METHOD WriteError
VAR_INPUT
	Event			: E_Event;
	Description 	: T_MaxString;
END_VAR
WriteEvent(ePriority_fault, Event, Description, TRUE);
//eState := E_ComponentState.eComponentState_error;
END_METHOD

METHOD WriteEvent
VAR_INPUT
	Priority		: E_Priority;
	Event			: E_Event;
	Description 	: T_MaxString;
	Signalize			: BOOL;
END_VAR
VAR
	tmpItem: ST_Event;
END_VAR
// chk
IF NOT __ISVALIDREF(fbEventLog) THEN
	RETURN;
END_IF

tmpItem.eComponent := eTyp;
tmpItem.eEventID := Event;
tmpItem.eMachineArea := eMachineArea;
tmpItem.ePriority := Priority;
tmpItem.nComponentID := iId;
tmpItem.sDescription := Description;
tmpItem.bSignalize := Signalize;

IF 	ptLastEvent <> 0 AND_THEN
	ptLastEvent^.bIsRaised AND_THEN
   	tmpItem.eEventID = ptLastEvent^.eEventID AND_THEN
	tmpItem.sDescription = ptLastEvent^.sDescription AND_THEN 
	tmpItem.ePriority = ptLastEvent^.ePriority THEN 
	RETURN;
END_IF

ptLastEvent := fbEventLog.SetEvent(tmpItem);
stLastEvent := tmpItem;
END_METHOD

METHOD WriteInfo
VAR_INPUT
	Event			: E_Event;
	Description 	: T_MaxString;
END_VAR
WriteEvent(ePriority_info, Event, Description, FALSE);
END_METHOD

METHOD WriteWarning
VAR_INPUT
	Event			: E_Event;
	Description 	: T_MaxString;
	Signal			: BOOL;
END_VAR
VAR
	tmpItem			: ST_Event;
END_VAR
WriteEvent(ePriority_warning, Event, Description, Signal);
END_METHOD

END_FUNCTION_BLOCK

// ---- BaseComponents/EventLog/FB_EventLog.TcPOU
/// HMI access provider (host for sub hmi provider)
FUNCTION_BLOCK  FB_EventLog
VAR	
	/// interfaces
	ILog						: ITFLoggingProvider;
	stLogConfig					: ST_LoggingConfig;
	
	/// Logging Provider
	fbDebugLog					: FB_DebugLoggingProvider;
	fbFileLog					: FB_FileLoggingProvider;
	fbEventLog					: FB_EventLoggingProvider;	
	fbEventlogger 				: FB_TcEventLogger;


	/// default notification array mirror (for compare)
	aEvents						: ARRAY[0..iMaxIdxEvents] OF ST_Event;
	aEventsMirror				: ARRAY[0..iMaxIdxEvents] OF ST_Event;
	diEventsChanged				: DINT;	
	diEventsChangedOld			: DINT;	
	nLastIndex					: INT;
	
	ptLastEvent					: POINTER TO ST_Event;
	
	//aEventsMirror				: ARRAY[0..iMaxIdxMachineAreas, 0..iMaxIdxComponent, 0..iMaxIdxEvents] OF ST_Event;
	/// private var's
	eErrorLevel					: E_Priority;
	eErrorLevelMirror			: E_Priority;	
	eLogLevel					: E_LogLevel;	
	
	bMute						: BOOL;
	
	fbAlarm						: FB_TcAlarm;
	fbMessage					: FB_TcMessage;
END_VAR

///
/// Event Log
/// Hannes Fuger /www.asma.at/01.2016
///

PROPERTY Config : ST_LoggingConfig
GET
Config := stLogConfig;
END_GET
SET
stLogConfig := Config;
END_SET
END_PROPERTY

/// System error level
PROPERTY ErrorLevel : E_Priority
GET // INTERNAL
ErrorLevel := eErrorLevel;
END_GET
END_PROPERTY

PROPERTY EventsChanged : BOOL
GET
EventsChanged := diEventsChanged <> diEventsChangedOld;
END_GET
END_PROPERTY

/// Filtert aktuelle Meldungen
METHOD PUBLIC FilterEvents : BOOL
VAR_INPUT
	/// Notification filter
	stFilter	: ST_EventFilter;
END_VAR
VAR_IN_OUT
	/// notification array (result)
	aResult		: ARRAY[0..iMaxIdxEvents] OF ST_Event;
END_VAR
VAR
	idx, iRes, iLast 		: INT;
	bFilterOk				: BOOL;
END_VAR
iRes := 0;
MEMSET(ADR(aResult), 0, SIZEOF(aResult));
iLast := nLastIndex+1;

FOR idx := 0 TO iMaxIdxEvents DO
	bFilterOk := TRUE;
	// IsRaised - Filter
	IF (stFilter.eIsRaisedFilter = eBoolFilter_false AND aEvents[iLast].bIsRaised) OR_ELSE 
	   (stFilter.eIsRaisedFilter = eBoolFilter_true AND NOT aEvents[iLast].bIsRaised) THEN
		bFilterOk := FALSE;
	END_IF
	
	// Area - Filter
	IF (stFilter.eAreaFilter <> E_MachineArea.eMachineArea_none) AND_THEN
	   (stFilter.eAreaFilter <> aEvents[iLast].eMachineArea) THEN
		bFilterOk := FALSE;
	END_IF
	
	// Error - Filter
	IF bFilterOk AND ((stFilter.eErrorFilter AND (aEvents[iLast].ePriority = ePriority_fault OR aEvents[iLast].ePriority = ePriority_faultEmergency OR aEvents[iLast].ePriority = ePriority_faultFastStop))
	// Warning - Filter
	OR (stFilter.eWarningFilter AND aEvents[iLast].ePriority = E_Priority.ePriority_warning)	
	// Info - Filter
	OR (stFilter.eInfoFilter AND aEvents[iLast].ePriority = E_Priority.ePriority_info)) THEN
		
		// add notification to result
		MEMCPY(ADR(aResult[iRes]), ADR(aEvents[iLast]), SIZEOF(aEvents[iLast]));
		iRes := iRes + 1;
	END_IF
	iLast := (iLast+1) MOD (iMaxIdxEvents+1);	
END_FOR

IF iRes > 0 THEN
	FilterEvents := TRUE;
END_IF
END_METHOD

PROPERTY LastIndex : INT
GET
LastIndex := nLastIndex;
END_GET
END_PROPERTY

PROPERTY Logger : REFERENCE TO ITFLoggingProvider
GET
Logger REF= ILog;
END_GET
END_PROPERTY

PROPERTY Mute : BOOL
GET
Mute := bMute;
END_GET
SET
bMute := Mute;
END_SET
END_PROPERTY

PROPERTY NextIndex : INT
GET
NextIndex := (nLastIndex+1) MOD (iMaxIdxEvents+1);
END_GET
END_PROPERTY

/// sets the corresponding notification item flag raised
{attribute 'object_name' := 'QuittAll'}
METHOD QuittAll
VAR_INPUT
	eMachineArea	: E_MachineArea;
END_VAR
VAR
	ni				: INT;
END_VAR
FOR ni := 0 TO iMaxIdxEvents DO	
	IF NOT aEvents[ni].bIsRaised THEN
		CONTINUE;
	END_IF
	
	IF aEvents[ni].eMachineArea = eMachineArea OR eMachineArea = E_MachineArea.eMachineArea_none THEN
		QuittEvent(	aEvents[ni]);
	END_IF
END_FOR
END_METHOD

/// sets the corresponding notification item flag raised
{attribute 'object_name' := 'QuittEvent'}
METHOD QuittEvent
VAR_INPUT
	stItem			: ST_Event;
END_VAR
VAR
	ni				: INT;
	cmpItem			: ST_Event;
END_VAR
// suchen ob ähnlicher Eintrag vorhanden 
// auch diesen quittieren

FOR ni := 0 TO iMaxIdxEvents DO	
	IF aEvents[ni].bIsRaised THEN
		cmpItem := 	aEvents[ni];
		// gleichsetzen damit beim Cmp kein Unterschied bei diesen Werten
		cmpItem.dtQuitTime := stItem.dtQuitTime;			
		cmpItem.dtRaiseTime := stItem.dtRaiseTime;	
		cmpItem.nIdx := stItem.nIdx;	
		
		IF MEMCMP(ADR(cmpItem), ADR(stItem), SIZEOF(ST_EVENT)) = 0 THEN
			aEvents[ni].bIsRaised := FALSE;
			aEvents[ni].dtQuitTime := Statics.dtNow;
			aEvents[ni].sQuitTime := SEL(aEvents[ni].dtQuitTime = DT#1970-01-01-00:00:00, REPLACE(DT_TO_STRING(aEvents[ni].dtQuitTime), '', 3, 1), '');		
		END_IF
		
	END_IF
END_FOR
END_METHOD

/// resets all notification flags and reset-needed state 
{attribute '' := ''}
{attribute 'object_name' := 'Reset'}
METHOD Reset
VAR
	ii: INT;
END_VAR
// reset all items in default notification array
MEMSET(ADR(aEvents), 0, SIZEOF(aEvents));
MEMSET(ADR(aEventsMirror), 0, SIZEOF(aEventsMirror));

// set default message priority
FOR ii := 0 TO iMaxIdxEvents DO
	aEvents[ii].ePriority := E_Priority.ePriority_fault;
END_FOR

nLastIndex := -1;

eErrorLevel			:= ePriority_none;
eErrorLevelMirror	:= ePriority_none;
eLogLevel			:= eLogLevelNone;

// set up logging provider
IF stLogConfig.eLoggingProvider = eLoggingProviderFile THEN
	fbFileLog(stLogConfig := stLogConfig);
	ILog := fbFileLog;
ELSIF stLogConfig.eLoggingProvider = eLoggingProviderEventLog THEN
	fbEventLog(stLogConfig := stLogConfig);
	ILog := fbEventLog;
ELSE // default
	ILog := fbDebugLog;
END_IF
END_METHOD

METHOD Run : E_ComponentState
VAR	/// private variabe
	ii			: INT;	
END_VAR
// run Logger
IF ILog <> 0 THEN
	ILog.Run();
END_IF

diEventsChangedOld := diEventsChanged;
// trigger notification changes
IF (MEMCMP(ADR(aEventsMirror), ADR(aEvents), SIZEOF(aEvents)) <> 0) THEN
	diEventsChanged := diEventsChanged  + 1; // in case of index-overrun, it (re)starts itself (-DINT max)
	aEventsMirror := aEvents;
END_IF

// get max error level
eErrorLevel := E_Priority.ePriority_none;
FOR ii := 0 TO iMaxIdxEvents DO	
	IF aEvents[ii].bIsRaised THEN
		eErrorLevel := MAX(eErrorLevel, aEvents[ii].ePriority);
		IF eErrorLevel <> eErrorLevelMirror THEN
			eErrorLevelMirror := eErrorLevel;
			CASE eErrorLevel OF
				E_Priority.ePriority_none,
				E_Priority.ePriority_info:
					eLogLevel := E_Loglevel.eLogLevelInformation;
				E_Priority.ePriority_warning:
					eLogLevel := E_Loglevel.eLogLevelWarning;
				E_Priority.ePriority_fault,
				E_Priority.ePriority_faultFastStop,
				E_Priority.ePriority_faultEmergency:
					eLogLevel := E_Loglevel.eLogLevelError;
			END_CASE
			ILog.AddLog(Concat6('ErrorLevel changed, ID: ', INT_TO_STRING(aEvents[ii].nComponentID),'-',INT_TO_STRING(aEvents[ii].eEventID),', MSG: ', aEvents[ii].sDescription), 'Supervision', eLogLevel);
		END_IF
	END_IF
END_FOR
END_METHOD

/// sets the corresponding notification item flag raised
{attribute 'object_name' := 'SetEvent'}
METHOD SetEvent : POINTER TO ST_Event
VAR_INPUT
	/// item to set
	stItem: ST_Event;
END_VAR
VAR
	tmpIndex		: INT;
	cmpItem			: ST_Event;
END_VAR
// suchen ob Eintrag schon vorhanden 
// nach gewisser zeit wieder eintragen
// sonst nichts unterenheme

// set item in default notification array 
tmpIndex := nextIndex;

// letzter Event der selbe?
IF tmpIndex > 0 THEN
	cmpItem := aEvents[LastIndex];
	// gleichsetzen damit beim Cmp kein Unterschied bei diesen Werten
	cmpItem.dtQuitTime := stItem.dtQuitTime;
	cmpItem.dtRaiseTime := stItem.dtRaiseTime;
	cmpItem.nIdx := stItem.nIdx;
	
	IF MEMCMP(ADR(stItem), ADR(cmpItem), SIZEOF(ST_Event)) = 0 THEN 
		RETURN;
	END_IF
END_IF


aEvents[tmpIndex] := stItem;
aEvents[tmpIndex].nIdx := tmpIndex;
aEvents[tmpIndex].bIsRaised := TRUE;
aEvents[tmpIndex].dtRaiseTime := Statics.dtNow;
aEvents[tmpIndex].dtQuitTime := StaticsConstant.dtMinValue;

aEvents[tmpIndex].sRaiseTime := SEL(aEvents[tmpIndex].dtRaiseTime = DT#1970-01-01-00:00:00, REPLACE(DT_TO_STRING(aEvents[tmpIndex].dtRaiseTime), '', 3, 1), '');
aEvents[tmpIndex].sQuitTime := SEL(aEvents[tmpIndex].dtQuitTime = DT#1970-01-01-00:00:00, REPLACE(DT_TO_STRING(aEvents[tmpIndex].dtQuitTime), '', 3, 1), '');

nLastIndex := tmpIndex;
SetEvent := ADR(aEvents[nLastIndex]);
END_METHOD

METHOD WriteError
VAR_INPUT
	Event			: E_Event;
	Description 	: T_MaxString;
END_VAR
WriteEvent(ePriority_fault, Event, Description, TRUE);
//eState := E_ComponentState.eComponentState_error;
END_METHOD

METHOD WriteEvent
VAR_INPUT
	Priority		: E_Priority;
	Event			: E_Event;
	Description 	: T_MaxString;
	Signalize		: BOOL;
END_VAR
VAR
	tmpItem			: ST_Event;
END_VAR
// chk

tmpItem.eComponent := E_ComponentType.eComponentType_none;
tmpItem.eEventID := Event;
tmpItem.eMachineArea := E_MachineArea.eMachineArea_common;
tmpItem.ePriority := Priority;
tmpItem.nComponentID := 0;
tmpItem.sDescription := Description;
tmpItem.bSignalize := Signalize;

IF 	ptLastEvent <> 0 AND_THEN
	ptLastEvent^.bIsRaised AND_THEN
   	tmpItem.eEventID = ptLastEvent^.eEventID AND_THEN
	tmpItem.sDescription = ptLastEvent^.sDescription AND_THEN 
	tmpItem.ePriority = ptLastEvent^.ePriority THEN 
	RETURN;
END_IF

ptLastEvent := SetEvent(tmpItem);
END_METHOD

METHOD WriteInfo
VAR_INPUT
	Event			: E_Event;
	Description 	: T_MaxString;
END_VAR
WriteEvent(ePriority_info, Event, Description, FALSE);
END_METHOD

METHOD WriteWarning
VAR_INPUT
	Event			: E_Event;
	Description 	: T_MaxString;
	Signal			: BOOL;
END_VAR
VAR
	tmpItem			: ST_Event;
END_VAR
WriteEvent(ePriority_warning, Event, Description, Signal);
END_METHOD

END_FUNCTION_BLOCK

// ---- Visualisation/P_Visu.TcPOU
PROGRAM P_Visu
VAR
	bFirstRun					: BOOL := TRUE;	
	
END_VAR

IF bFirstRun THEN
	bFirstRun := FALSE;
	FirstRun();
END_IF

JogButton();
SwitchButton();
SyncVariable();

METHOD FirstRun : BOOL
VAR_INPUT
END_VAR
GVL_VISU.stMachineConfig := P_Machine.MachineConfig;	
GVL_VISU.stCurMat := fbmat.Mat;
END_METHOD

METHOD JogButton : BOOL
VAR_INPUT
END_VAR
// JOG X
IF GVL_VISU.stMaintCmds.bJogXBw THEN
	GVL.fbMatAndToolHandling.JogX(TRUE);
ELSIF GVL_VISU.stMaintCmds.bJogXFw THEN
	GVL.fbMatAndToolHandling.JogX(FALSE);
ELSE
	GVL.fbMatAndToolHandling.JogXStop();
END_IF

// JOG Y
IF GVL_VISU.stMaintCmds.bJogYBw THEN
	GVL.fbMatAndToolHandling.JogY(TRUE);
ELSIF GVL_VISU.stMaintCmds.bJogYFw THEN
	GVL.fbMatAndToolHandling.JogY(FALSE);
ELSE
	GVL.fbMatAndToolHandling.JogYStop();
END_IF

// JOG Punch
IF GVL_VISU.stMaintCmds.bJogPunchBw THEN
	GVL.fbPunchEngine.Jog(FALSE, TRUE);
ELSIF GVL_VISU.stMaintCmds.bJogPunchFw THEN
	GVL.fbPunchEngine.Jog(TRUE, FALSE);
ELSE
	GVL.fbPunchEngine.JogStop();
END_IF

// JOG BELT
IF GVL_VISU.stMaintCmds.bJogOutletBelt THEN
	GVL.fbPunchEngine.OutletBeltJog(TRUE);
ELSE
	GVL.fbPunchEngine.OutletBeltJog(FALSE);
END_IF
END_METHOD

METHOD SwitchButton : BOOL
VAR_STAT
	stNullPunchCmds				: ST_PunchCmds;
	stNullMaintCmds				: ST_MaintCmds;
END_VAR
// PUNCH COMMANDS
IF MEMCMP(ADR(GVL_VISU.stPunchCmds), ADR(stNullPunchCmds), SIZEOF(ST_PunchCmds)) <> 0 THEN
	IF GVL_VISU.stPunchCmds.bLoad THEN
		P_Machine.LoadMat(GVL_VISU.stCurMat);		
		P_Machine.LoadJob(GVL_VISU.stPunchJob);	
	END_IF
	
	IF GVL_VISU.stPunchCmds.bStart THEN	
		P_Machine.LoadMat(GVL_VISU.stCurMat);	
		P_Machine.Start(GVL_VISU.stPunchJob);	
	END_IF
	
	IF GVL_VISU.stPunchCmds.bStop THEN
		P_Machine.Stop();	
	END_IF
	
	IF GVL_VISU.stPunchCmds.bResume THEN
		P_Machine.Resume();	
	END_IF
	
	IF GVL_VISU.stPunchCmds.bHalt THEN
		P_Machine.ClearJob();
		P_Machine.Halt();	
	END_IF	
		
	IF GVL_VISU.stPunchCmds.bLoadLeft THEN
		P_Machine.Maint(TRUE, TRUE, FALSE);	
	END_IF	
	
	IF GVL_VISU.stPunchCmds.bLoadRight THEN
		P_Machine.Maint(TRUE, TRUE, TRUE);	
	END_IF	
	
	IF GVL_VISU.stPunchCmds.bLoadStop THEN
		P_Machine.Halt();	
	END_IF	
	
	IF GVL_VISU.stPunchCmds.bUnlock THEN
		IF fbSafetyLock.Locked THEN
			GVL.fbSafetyLock.Unlock();
		ELSE
			GVL.fbSafetyLock.Lock();
		END_IF
	END_IF		
	
	IF GVL_VISU.stPunchCmds.bMoveTDC THEN
		GVL.fbPunchEngine.MoveTDC();	
	END_IF	
	
	IF GVL_VISU.stPunchCmds.bOutletBelt THEN
		GVL.fbPunchEngine.OutletBeltOnce();	
	END_IF	
		
	IF GVL_VISU.stPunchCmds.bOverride THEN
		P_Machine.Override := GVL_VISU.stPunchParam.fOverride;
	END_IF	
END_IF

// RESET PUNCH COMMANDS
GVL_VISU.stPunchCmds.bLoad := FALSE;
GVL_VISU.stPunchCmds.bStart := FALSE;
GVL_VISU.stPunchCmds.bStop := FALSE;
GVL_VISU.stPunchCmds.bResume := FALSE;
GVL_VISU.stPunchCmds.bHalt := FALSE;
GVL_VISU.stPunchCmds.bLoadLeft := FALSE;
GVL_VISU.stPunchCmds.bLoadRight := FALSE;
GVL_VISU.stPunchCmds.bMoveTDC := FALSE;
GVL_VISU.stPunchCmds.bOutletBelt := FALSE;
GVL_VISU.stPunchCmds.bOverride := FALSE;
GVL_VISU.stPunchCmds.bUnlock := FALSE;
GVL_VISU.stPunchCmds.bLoadStop := FALSE;

// MAINT COMMANDS
IF MEMCMP(ADR(GVL_VISU.stMaintCmds), ADR(stNullMaintCmds), SIZEOF(ST_MaintCmds)) <> 0 THEN	
	IF GVL_VISU.stMaintCmds.bLoadConfig THEN
		P_Machine.LoadConfig(GVL_VISU.stMachineConfig);
	END_IF
	
	IF GVL_VISU.stMaintCmds.bChangeTool THEN
		GVL.fbMatAndToolHandling.ChangeTool(GVL_VISU.stMaintParam.nChangeTool);
	END_IF
	
	IF GVL_VISU.stMaintCmds.bMoveXYMaint THEN
		P_Machine.Maint(TRUE, TRUE, FALSE);	
	END_IF
	
	IF GVL_VISU.stMaintCmds.bMoveXYMaintAlt THEN
		P_Machine.Maint(TRUE, TRUE, TRUE);	
	END_IF
	
	IF GVL_VISU.stMaintCmds.bReset THEN
		P_Machine.Reset();	
	END_IF	
	
	IF GVL_VISU.stMaintCmds.bMovePunchTDC THEN
		GVL.fbPunchEngine.MoveTDC();	
	END_IF	
	
	IF GVL_VISU.stMaintCmds.bSetZero THEN
		GVL.fbPunchEngine.SetZeroOffset();	
	END_IF	
	
END_IF

// RESET MAINT COMMANDS
GVL_VISU.stMaintCmds.bLoadConfig := FALSE;
GVL_VISU.stMaintCmds.bChangeTool := FALSE;
GVL_VISU.stMaintCmds.bMoveXYMaint := FALSE;
GVL_VISU.stMaintCmds.bMoveXYMaintAlt := FALSE;
GVL_VISU.stMaintCmds.bReset := FALSE;
GVL_VISU.stMaintCmds.bMovePunchTDC := FALSE; 
GVL_VISU.stMaintCmds.bSetZero := FALSE;
END_METHOD

METHOD SyncVariable : BOOL
VAR_INPUT
END_VAR
// VISU TO PLC
stPunchInfo.sCleartext 				:= P_Machine.seqOpMode.ClearText;
stPunchInfo.nCurMat 				:= P_Machine.CurMat + 1;
stPunchInfo.nCurPunch 				:= P_Machine.CurPunch + 1;
stPunchInfo.nCurRun 				:= P_Machine.CurRun + 1;
stPunchInfo.nMaxPunches 			:= P_Machine.MaxPunch + 1;
stPunchInfo.nCountRemainHolesOfJob 	:= P_Machine.CountRemainHolesOfJob + 1;
stPunchInfo.nCountAllHolesOfJob 	:= P_Machine.CountAllHolesOfJob + 1;
stPunchInfo.nRemainTimeOfJob 		:= P_Machine.RemainTimeOfJob;
stPunchInfo.stCoordinate 			:= P_Machine.stCoordinate;
stPunchInfo.bPunching 				:= P_Machine.Punching;
stPunchInfo.bResumeAllowed 			:= P_Machine.ResumeAllowed;
stPunchInfo.eJobState 				:= P_Machine.JobState;
stPunchInfo.fOverride 				:= P_Machine.Override;
stPunchInfo.fPunchspeed				:= fbPunchEngine.fbPunchAxis.Velocity;
stPunchInfo.bLocked					:= fbSafetyLock.Locked;

// X - Axis
stMaintInfo.bXHomed					:= fbMatAndToolHandling.fbAxisX.Homed;
stMaintInfo.bXError					:= fbMatAndToolHandling.fbAxisX.Error;
stMaintInfo.bXMoving				:= fbMatAndToolHandling.fbAxisX.Moving;
stMaintInfo.fXPosition				:= fbMatAndToolHandling.fbAxisX.ActPos;
stMaintInfo.fXTemp					:= fbMatAndToolHandling.fbAxisX.AmplifierTemp;
stMaintInfo.fXMotorTemp				:= fbMatAndToolHandling.fbAxisX.MotorTemp;
                            		   
// Y - Axis                 		   
stMaintInfo.bYHomed					:= fbMatAndToolHandling.fbAxisY.Homed;        
stMaintInfo.bYError					:= fbMatAndToolHandling.fbAxisY.Error;        
stMaintInfo.bYMoving				:= fbMatAndToolHandling.fbAxisY.Moving;       
stMaintInfo.fYPosition				:= fbMatAndToolHandling.fbAxisY.ActPos;       
stMaintInfo.fYTemp					:= fbMatAndToolHandling.fbAxisY.AmplifierTemp;
stMaintInfo.fYMotorTemp				:= fbMatAndToolHandling.fbAxisY.MotorTemp;    
                            		   
// Punch - Axis             		   
stMaintInfo.bPunchHomed				:= fbPunchEngine.fbPunchAxis.Homed;        
stMaintInfo.bPunchError				:= fbPunchEngine.fbPunchAxis.Error;        
stMaintInfo.bPunchMoving			:= fbPunchEngine.fbPunchAxis.Moving;       
stMaintInfo.fPunchPosition			:= fbPunchEngine.fbPunchAxis.ActModuloPos;       
stMaintInfo.fPunchTemp				:= fbPunchEngine.fbPunchAxis.AmplifierTemp;
stMaintInfo.fPunchMotorTemp			:= fbPunchEngine.fbPunchAxis.MotorTemp;   
 
// ToolChanger              		   
stMaintInfo.bToolError				:= fbMatAndToolHandling.fbToolSelector.State = E_ComponentState.eComponentState_error;
stMaintInfo.bToolChanged			:= fbMatAndToolHandling.ToolChanged;
stMaintInfo.nToolSelect				:= fbMatAndToolHandling.CurTool;
                            		   
// Machine                  		   
stMaintInfo.bSequenceError			:= P_Machine.seqOpMode.State = E_SequenceState.eSequenceState_error;
stMaintInfo.bSafetyOk				:= fbSafety.SafetyOk;
stMaintInfo.bEmergency				:= NOT fbSafety.bNotHaltOk;
stMaintInfo.nPunchCount				:= fbPunchEngine.PunchCount;                         		  
stMaintInfo.nStep					:= P_Machine.seqOpMode.Step;
stMaintInfo.nSequence				:= P_Machine.seqOpMode.SequenceId;
//stMaintInfo.bSafetyDoor				:= ;

// PLC TO VISU
P_Machine.CheckPosBeforeRun 		:= GVL_VISU.stPunchParam.bCheckPosBeforeRun;
END_METHOD

END_PROGRAM

// ---- BaseComponents/Safety/FB_Safety.TcPOU
/// Function block for TwinSAFE communication.
FUNCTION_BLOCK FB_Safety EXTENDS FB_ComponentBase
VAR_OUTPUT	
	/// Quittieren Safety erforderlich	
	bSafetyQuittRequest		:BOOL;
	
	/// Not-Halt Status OK
	bNotHaltOk				:BOOL;
END_VAR
VAR
	/// IO reference
	stIn					: REFERENCE TO ST_SafetyIn;
	stOut					: REFERENCE TO ST_SafetyOut;
	/// private var's
	nStep					: INT;
	tonDelay				: TON;
	
	bSafetyOK				: BOOL;
	
END_VAR

METHOD FB_init : BOOL
VAR_INPUT
	bInitRetains : BOOL; // if TRUE, the retain variables are initialized (warm start / cold start)
	bInCopyCode : BOOL;  // if TRUE, the instance afterwards gets moved into the copy code (online change)
END_VAR
eTyp := E_ComponentType.eComponentType_Safety;
END_METHOD

/// resets TwinSAFE
{attribute 'object_name' := 'Reset'}
METHOD Reset
VAR
	ii: INT;
END_VAR
// base logic run
SUPER^.Reset();

tonDelay(IN := FALSE);
eState := E_ComponentState.eComponentState_resetting;
END_METHOD

/// Run component logic
{attribute 'object_name' := 'Run'}
METHOD Run : E_ComponentState
VAR
END_VAR
// base logic run
Run := SUPER^.Run();

IF NOT __ISVALIDREF(stIn) OR NOT __ISVALIDREF(stOut) THEN
	RETURN;
END_IF

stOut.bSAFE_NotHalt_Ok := stIn.bSAFE_NotHalt_Ok;
stOut.bRun_stop := TRUE;

// Anforderung zum quittieren der Sicherheit				
bSafetyQuittRequest := NOT stIn.bSAFE_NotHalt_Ok OR
						stIn.bSAFE_CommErr OR
						stIn.bSAFE_FbErr;

bNotHaltOk := stIn.bSAFE_NotHalt_Ok;
bSafetyOK := NOT stIn.bSAFE_CommErr AND NOT stIn.bSAFE_FbErr AND bNotHaltOk;

CASE nStep OF
	0: 	
		sClearText := 'wait for reset command.';
		IF stIn.bSAFE_CommErr THEN
			WriteError(eEvent_safetyError, 'TwinSAFE COM Error');
		ELSIF stIn.bSAFE_FbErr THEN
			WriteError(eEvent_safetyError, 'TwinSAFE FB Error');
		ELSIF NOT stIn.bSAFE_NotHalt_Ok THEN
			WriteError(eEvent_safetyError, 'TwinSAFE Not-Halt');
		END_IF		
		
		IF eState = E_ComponentState.eComponentState_resetting THEN  // -> in Reset() METHOD		
			stOut.bErrAckSafety_General := TRUE;
			nStep := 10;
		END_IF		
		
	10:	
		sClearText := 'Error ack TwinSAFE reset General';
		tonDelay(IN := TRUE, PT := T#1S);
		IF tonDelay.Q THEN
			stOut.bErrAckSafety_General := FALSE;
			tonDelay(IN := FALSE);
			IF stIn.bSAFE_FbErr OR stIn.bSAFE_CommErr OR NOT stIn.bSAFE_NotHalt_Ok THEN // chk error still active
				nStep := 0;
			ELSE
				stOut.bErrAckSafety_Drive := TRUE;
				nStep := 20;
			END_IF			
		END_IF
		
	20:	
		sClearText := 'Error ack TwinSAFE reset Drives';
		tonDelay(IN := TRUE, PT := T#1S);
		IF tonDelay.Q THEN
			stOut.bErrAckSafety_Drive := FALSE;
			tonDelay(IN := FALSE);
			nStep := 100;
		END_IF
		
	100:
		sClearText := 'Reset TwinSAFE Done';
		eState := E_ComponentState.eComponentState_running;
		nStep := 0;
		
END_CASE
END_METHOD

PROPERTY SafetyOk : BOOL
GET
SafetyOK := bSafetyOK;
END_GET
END_PROPERTY

/// Dependency injection method.
{attribute 'object_name' := 'SetReferences'}
METHOD INTERNAL SetReferences
VAR_IN_OUT
	/// IO reference
	stIORef: ST_SafetyIO;	
END_VAR
/// set up references
stIn REF= stIORef.stIn;
stOut REF= stIORef.stOut;
END_METHOD

END_FUNCTION_BLOCK

// ---- BaseComponents/EtherCAT/FB_EtherCATBus.TcPOU
FUNCTION_BLOCK FB_EtherCATBus EXTENDS FB_ComponentBase

VAR
	/// IO structure
	stIO 				: REFERENCE TO ST_EtherCatIO;
	oldEtherCATState	: INT;
	n3072Err			: INT;
END_VAR

///
/// EtherCAT driver.
/// Hannes Fuger / asma.at / 12.2015
///

METHOD FB_init : BOOL
VAR_INPUT
	bInitRetains : BOOL; // if TRUE, the retain variables are initialized (warm start / cold start)
	bInCopyCode : BOOL;  // if TRUE, the instance afterwards gets moved into the copy code (online change)
END_VAR
eTyp := E_ComponentType.eComponentType_EtherCAT;
END_METHOD

METHOD Run : E_ComponentState
VAR_INPUT
END_VAR
// base logic run
Run := SUPER^.Run();

// chk reference
IF NOT __ISVALIDREF(fbEventLog) THEN
	RETURN;
END_IF

IF oldEtherCATState = stIo.eEtherCATState THEN
	RETURN;
ELSE
	oldEtherCATState := stIo.eEtherCATState;
END_IF



// switch EtherCAT State
CASE stIO.eEtherCATState OF
	/// Link error
	eEtherCATState_LinkError :
		WriteError(eEvent_hardwareError, 'EtherCAT: Link error');
		
	/// I/O locked after link error (I/O reset required)
	eEtherCATState_IoLockedAfterLinkErr :
		WriteError(eEvent_hardwareError, 'EtherCAT: I/O locked after link error (I/O reset required)');
	
	/// Link error (redundancy adapter)
	eEtherCATState_LinkErrRedAdapter :
		WriteError(eEvent_hardwareError, 'EtherCAT: Link error (redundancy adapter)');
	
	/// Missing one frame (redundancy mode)
	eEtherCATState_MissingFrame :
		WriteError(eEvent_hardwareError, 'EtherCAT: Missing one frame (redundancy mode)');
	
	/// Out of send resources (I/O reset required)
	eEtherCATState_OutOfSendResources :
		WriteError(eEvent_hardwareError, 'EtherCAT: Out of send resources (I/O reset required)');
	
	/// Watchdog triggered
	eEtherCATState_WatchdogTriggered :
		WriteError(eEvent_hardwareError, 'EtherCAT: Watchdog triggered');
	
	/// Ethernet driver (miniport) not found
	eEtherCATState_EthernetDrvNotFound :
		WriteError(eEvent_hardwareError, 'EtherCAT: Ethernet driver (miniport) not found');
	
	/// I/O reset active
	eEtherCATState_IO_resetActive :
		WriteError(eEvent_hardwareError, 'EtherCAT: I/O reset active');
	
	/// At least one device in 'INIT' state
	eEtherCATState_AtLeastOneDeviceInit :
		WriteError(eEvent_hardwareError, 'EtherCAT: At least one device in INIT state');
	
	///  At least one device in 'PRE-OP' state
	eEtherCATState_AtLeastOneDevicePreOp :
		WriteError(eEvent_hardwareError, 'EtherCAT: At least one device in PRE-OP state');
	
	/// At least one device in 'SAFE-OP' state
	eEtherCATState_AtLeastOneDeviceSafeOp :
		WriteError(eEvent_hardwareError, 'EtherCAT: At least one device in SAFE-OP state');
	
	/// At least one device indicates an error state
	eEtherCATState_AtLeastOneDeviceError :
		WriteError(eEvent_hardwareError, 'EtherCAT: At least one device indicates an error state');
	
	/// DC not in sync
	eEtherCATState_DC_notInSync :
		WriteError(eEvent_hardwareError, 'EtherCAT: DC not in sync');

	ELSE // default 
		IF stIO.eEtherCATState = 1024 THEN
			n3072Err := n3072Err + 1;
		ELSIF stIO.eEtherCATState = 3072 THEN
			n3072Err := n3072Err + 1;
		ELSIF stIO.eEtherCATState <> 0 THEN
			WriteError(eEvent_hardwareError, Concat('EtherCAT Error: ', INT_TO_STRING(stIO.eEtherCATState)));
		END_IF
	
END_CASE
END_METHOD

/// Dependency injection method.
{attribute 'object_name' := 'SetReferences'}
METHOD SetReferences
VAR_IN_OUT
	/// IO structure
	stRefIO		: ST_EtherCatIO;
END_VAR
/// set up references
stIO REF= stRefIO;
END_METHOD

END_FUNCTION_BLOCK

// ---- BaseComponents/Supervision/FB_Supervision.TcPOU
/// Supervision function block - system watchdog
FUNCTION_BLOCK INTERNAL FB_Supervision EXTENDS FB_ComponentBase

VAR
	//aCodeError						: REFERENCE TO ARRAY[0..eCodeError_maxIdx] OF BOOL;
END_VAR

/// 
/// supervision function block of the project
/// TP/www.rmth.at/11.2014
/// 

//ToDo: run supervision (ES, Safety signals, IO-errors, etc.)

METHOD FB_init : BOOL
VAR_INPUT
	bInitRetains : BOOL; // if TRUE, the retain variables are initialized (warm start / cold start)
	bInCopyCode : BOOL;  // if TRUE, the instance afterwards gets moved into the copy code (online change)
END_VAR
eTyp := E_ComponentType.eComponentType_Supervision;
END_METHOD

/// resets all notification flags and reset-needed state 
{attribute '' := ''}
{attribute 'object_name' := 'Reset'}
METHOD Reset
VAR
	ii: INT;
END_VAR
// base logic run
SUPER^.Reset();

// reset code errors
MEMSET(ADR(GVL_Supervision.aCodeErr), 0, SIZEOF(GVL_Supervision.aCodeErr));
END_METHOD

/// Run component logic
{attribute 'object_name' := 'Run'}
METHOD Run : E_ComponentState
VAR
	ii			: INT;
END_VAR
// base logic run
Run := SUPER^.Run();

// chk reference
IF NOT __ISVALIDREF(fbEventLog) THEN //OR NOT __ISVALIDREF(aCodeError) THEN
	RETURN;
END_IF

//ToDo: run supervision (ES, Safety signals, IO-errors, etc.)

// task cycle time exceeded
IF Statics.stPlcSystemInfo.stPlcTaskSystemInfo.CycleTimeExceeded THEN
	WriteError(eEvent_systemError, 'Cycletime exceeded');
END_IF

// check for code errors
IF GVL_Supervision.aCodeErr[eCodeError_bounds] THEN
	WriteError(eEvent_systemError, 'Code error: check bounds.');
	
ELSIF GVL_Supervision.aCodeErr[eCodeError_divDInt] THEN
	WriteError(eEvent_systemError, 'Code error: check div int.');
	
ELSIF GVL_Supervision.aCodeErr[eCodeError_divLInt] THEN
	WriteError(eEvent_systemError, 'Code error: check div lint.');
	
ELSIF GVL_Supervision.aCodeErr[eCodeError_divLReal] THEN
	WriteError(eEvent_systemError, 'Code error: check div lreal.');
	
ELSIF GVL_Supervision.aCodeErr[eCodeError_divReal] THEN
	WriteError(eEvent_systemError, 'Code error: check div real.');
	
ELSIF GVL_Supervision.aCodeErr[eCodeError_pointer] THEN
	WriteError(eEvent_systemError, 'Code error: check pointer.');
	
ELSIF GVL_Supervision.aCodeErr[eCodeError_rangeSigned] THEN
	WriteError(eEvent_systemError, 'Code error: check range signed.');
	
ELSIF GVL_Supervision.aCodeErr[eCodeError_rangeUnsigned] THEN
	WriteError(eEvent_systemError, 'Code error: check range usigned.');
	
END_IF
END_METHOD

END_FUNCTION_BLOCK

// ---- BaseComponents/SafetyLockDriver/FB_SafetyLock.TcPOU
/// Saftey Lock driver.
FUNCTION_BLOCK FB_SafetyLock EXTENDS FB_ComponentBase

VAR
	/// IO structure
	stIn 				: REFERENCE TO ST_SafetyLockIn;
	stOut 				: REFERENCE TO ST_SafetyLockOut;
END_VAR

///
/// Saftey Lock driver.
/// Hannes Fuger @ asma.at		/ 09.2015
///

PROPERTY Closed : BOOL
GET
Closed := not stIn.bSaftyOK;
END_GET
END_PROPERTY

METHOD FB_init : BOOL
VAR_INPUT
	bInitRetains : BOOL; // if TRUE, the retain variables are initialized (warm start / cold start)
	bInCopyCode : BOOL;  // if TRUE, the instance afterwards gets moved into the copy code (online change)
END_VAR
eTyp := E_ComponentType.eComponentType_SafetyLock;
END_METHOD

METHOD Lock
VAR_INPUT
END_VAR
//cmd
stOut.bLock := TRUE;
END_METHOD

PROPERTY Locked : BOOL
GET
Locked := stIn.bSaftyOK AND stOut.bLock;
END_GET
END_PROPERTY

PROPERTY Opened : BOOL
GET
Opened := NOT stIn.bSaftyOK;
END_GET
END_PROPERTY

PROPERTY Referenced : BOOL
GET
Referenced:= __ISVALIDREF(stIn) AND __ISVALIDREF(stout);
END_GET
END_PROPERTY

/// Run component logic
{attribute 'object_name' := 'Run'}
METHOD Run : E_ComponentState
VAR
END_VAR
// base logic run
Run := SUPER^.Run();

stOut.bSaftyOk := stin.bSaftyOK;
END_METHOD

PROPERTY SafetyOk : BOOL
GET
SafetyOk := stIn.bSaftyOK;
END_GET
END_PROPERTY

PROPERTY SafetyOkAdr : POINTER TO BOOL
GET
SafetyOkAdr := ADR(stIn.bSaftyOK);
END_GET
END_PROPERTY

/// Set IO reference
{attribute 'object_name' := 'SetReferences'}
METHOD SetReferences
VAR_IN_OUT
	/// IO structure
	stRefIO 	: ST_SafetyLockIO;
END_VAR
stIn REF= stRefIO.stIn;
stOut REF= stRefIO.stOut;
END_METHOD

METHOD Unlock
VAR_INPUT
END_VAR
//cmd
stOut.bLock := FALSE;
END_METHOD

END_FUNCTION_BLOCK

// ---- Components/Mat/FB_Mat.TcPOU
FUNCTION_BLOCK FB_Mat EXTENDS FB_Componentbase

VAR
	// Reference of Mat
	stMat						: ST_Mat;
	
	// Coordinates of Mat
	nRunNr						: UINT;
	eCoordinatesSortState		: E_CoordinatesSortState;
	stCoordinates				: ARRAY[0..MATHOLES_COUNT] OF ST_Coordinate;
	nCorrdinatesCount			: UDINT;

END_VAR

METHOD Cmp_Coordinates : INT
VAR_INPUT
	ptFirst				: POINTER TO ST_Coordinate;
	ptSecond			: POINTER TO ST_Coordinate;
END_VAR
IF ptFirst = 0 OR ptSecond = 0 THEN
	RETURN;
END_IF

Cmp_Coordinates := 0;

IF ptFirst^.fX > ptSecond^.fX THEN
	Cmp_Coordinates := 1;
	
ELSIF ptFirst^.fX < ptSecond^.fX THEN
	Cmp_Coordinates := -1;	
	
ELSIF ptFirst^.fX = ptSecond^.fX THEN
	IF ptFirst^.fY > ptSecond^.fY THEN
		Cmp_Coordinates := 1;	
		
	ELSIF ptFirst^.fY < ptSecond^.fY THEN
		Cmp_Coordinates := -1;	
		
	END_IF
END_IF
END_METHOD

METHOD ConvertRun : E_OperationResult
VAR_INPUT
	Run						: UINT;
END_VAR
/// CHECK REFERENCES
ConvertRun := E_OperationResult.eOperationResult_NOk;

// check mat and Run definitions 
IF NOT stMat.astRuns[Run].bActive THEN
	RETURN;
END_IF

nRunNr := Run;

/// RESET OLD VALUES
MEMSET(ADR(stCoordinates), 0, SIZEOF(stCoordinates));
nCorrdinatesCount := HolesOfRun(Run, ADR(stCoordinates));
eCoordinatesSortState := E_CoordinatesSortState.eCoordinatesSortState_unsorted;

IF nCorrdinatesCount > 0 THEN
	ConvertRun := E_OperationResult.eOperationResult_Ok;
END_IF
END_METHOD

METHOD Count_HolesOfElement :  UDINT
VAR_INPUT
	Run						: UINT;
	Element					: UINT;
END_VAR

VAR
	tmpRun					: REFERENCE TO ST_MatRun;
	tmpElement				: REFERENCE TO ST_Element;
	
	tmpCount				: UDINT;
END_VAR
/// GET ELEMENT CHECK REFERENZES
//IF NOT __ISVALIDREF(refMat) THEN	RETURN;	END_IF 
tmpRun REF= stMat.astRuns[Run];
IF NOT __ISVALIDREF(tmpRun) THEN	RETURN;	END_IF
tmpElement REF= tmpRun.astElements[Element];
IF NOT __ISVALIDREF(tmpElement) THEN	RETURN;	END_IF

/// CALCULATE HOLES

IF NOT tmpElement.bActive THEN	
	Count_HolesOfElement := 0;
	RETURN;	
END_IF

tmpCount :=  tmpElement.nCountX * tmpElement.nCountY;
 
IF tmpElement.bMirroring THEN
	tmpCount := tmpCount*2;
END_IF

Count_HolesOfElement := tmpCount;
END_METHOD

METHOD Count_HolesOfRun :  UDINT
VAR_IN_OUT
	Run						: UINT;
END_VAR

VAR
	tmpCount				: UDINT;
	ni						: UINT;
END_VAR
/// CHECK REFERENZES
//IF NOT __ISVALIDREF(refMat) THEN	RETURN;	END_IF 

IF NOT stMat.astRuns[Run].bActive THEN
	Count_HolesOfRun := 0;	
	RETURN;
END_IF

FOR ni := 0 TO MATELEMENTS_COUNT DO
	tmpCount := tmpCount + Count_HolesOfElement(Run, ni);
END_FOR

Count_HolesOfRun := tmpCount;
END_METHOD

METHOD FB_init : BOOL
VAR_INPUT
	bInitRetains : BOOL; // if TRUE, the retain variables are initialized (warm start / cold start)
	bInCopyCode : BOOL;  // if TRUE, the instance afterwards gets moved into the copy code (online change)
END_VAR
eTyp := E_ComponentType.eComponentType_Mat;
END_METHOD

METHOD GetCoordinate : E_OperationResult
VAR_INPUT
	RunNr					: UINT;
	IndexNr					: UDINT;
	ptCoordinate			: POINTER TO ST_Coordinate;
END_VAR
GetCoordinate := E_OperationResult.eOperationResult_NOk;

IF IndexNr > nCorrdinatesCount THEN
	RETURN;
END_IF

IF eCoordinatesSortState =  E_CoordinatesSortState.eCoordinatesSortState_unsorted OR
	eCoordinatesSortState =  E_CoordinatesSortState.eCoordinatesSortState_undefined THEN
	RETURN;
END_IF

IF RunNr <> nRunNr THEN
	RETURN;
END_IF

ptCoordinate^ := stCoordinates[IndexNr];

GetCoordinate := E_OperationResult.eOperationResult_Ok;
END_METHOD

METHOD HolesOfElement : UDINT
VAR_INPUT
	Run						: UINT;
	Element					: UINT;
	ptArray					: POINTER TO ARRAY[0..MATHOLES_COUNT] OF ST_Coordinate;
END_VAR

VAR
	tmpRun					: REFERENCE TO ST_MatRun;
	tmpElement				: REFERENCE TO ST_Element;
	tmptool					: REFERENCE TO ST_Tool;
	tmptoolholder			: REFERENCE TO ST_Toolholder;
	
	tmpCount				: UDINT;
	tmpX_Pos				: REAL;
	tmpY_Pos				: REAL;
	tmpX_PosFirst			: REAL;
	tmpY_PosFirst			: REAL;
	
	tmpArrayIdx				: UINT;
	ni, nj					: UINT;
	
END_VAR
IF ptArray = 0 THEN
	RETURN;
END_IF

MEMSet(ptArray,0,SIZEOF(POINTER TO ARRAY[0..MATHOLES_COUNT] OF ST_Coordinate));

/// DEFINE VARIABLES, CHECK REFERENZES	
//IF NOT __ISVALIDREF(refMat) THEN	RETURN;	END_IF 

tmpRun REF= stMat.astRuns[Run];
IF NOT __ISVALIDREF(tmpRun) THEN	RETURN;	END_IF

tmpElement REF= tmpRun.astElements[Element];
IF NOT __ISVALIDREF(tmpElement) THEN	RETURN;	END_IF

tmpTool REF= tmpRun.stTool;
tmpToolholder REF= tmpRun.stToolHolder;
IF NOT __ISVALIDREF(tmpTool) OR NOT __ISVALIDREF(tmpToolholder)	THEN	RETURN;	END_IF

HolesOfElement := tmpCount := Count_HolesOfElement(Run, Element);
IF tmpCount <= 0 OR tmpCount > MATHOLES_COUNT THEN	RETURN;	END_IF

/// SET ZERO IF NOT MULTIDIE
IF NOT tmpToolholder.bMultiDie THEN
	tmpToolholder.nDieCount := 0;
END_IF	

/// CALCULATE COORDINATES OF FIRST HOLE
IF tmpElement.bCentering THEN
	tmpX_PosFirst := tmpElement.fX_Pos;
	tmpY_PosFirst := (stMat.fWidth - (tmpToolholder.fDie_Offset * (tmpToolholder.nDieCount - 1) + tmpElement.fDistanceY * (tmpElement.nCountY - 1))) / 2;
ELSE           
	tmpX_PosFirst := tmpElement.fX_Pos;
	tmpY_PosFirst:= tmpElement.fY_Pos;
END_IF


/// CALCULATE ARRAY
tmpArrayIdx := 0;

FOR ni := 0 TO tmpElement.nCountX-1 DO
	FOR nj:= 0 TO tmpElement.nCountY-1 DO
		
		CASE tmpElement.eOrigin OF
			
			E_ElementOrigin.eElementOrigin_ButtomRight:
				tmpX_Pos := tmpX_PosFirst + ni*tmpElement.fDistanceX;	
				tmpY_Pos := tmpY_PosFirst + nj*tmpElement.fDistanceY;		
		
			E_ElementOrigin.eElementOrigin_ButtomLeft:	
				tmpX_Pos := stMat.fLenght - (tmpX_PosFirst + ni*tmpElement.fDistanceX);	
				tmpY_Pos := tmpY_PosFirst + nj*tmpElement.fDistanceY;		
					
			E_ElementOrigin.eElementOrigin_TopRight:
				tmpX_Pos := tmpX_PosFirst + ni*tmpElement.fDistanceX;	
				tmpY_Pos := stMat.fWidth - (tmpY_PosFirst + nj*tmpElement.fDistanceY) - (tmpToolholder.fDie_Offset * (tmpToolholder.nDieCount - 1)) ;	
					
			E_ElementOrigin.eElementOrigin_TopLeft:
				tmpX_Pos := stMat.fLenght - (tmpX_PosFirst + ni*tmpElement.fDistanceX);	
				tmpY_Pos := stMat.fWidth - (tmpY_PosFirst + nj*tmpElement.fDistanceY) - (tmpToolholder.fDie_Offset * (tmpToolholder.nDieCount - 1)) ;	
		
		END_CASE
		
		/// ADD OFFEST OF TOOLHOLDER
		ptArray^[tmpArrayIdx].fX := tmpX_Pos + tmpToolholder.fX_Offset;
		ptArray^[tmpArrayIdx].fY := tmpY_Pos + tmpToolholder.fY_Offset;		
		tmpArrayIdx := tmpArrayIdx + 1;		
		
	END_FOR
END_FOR
END_METHOD

METHOD HolesOfRun : UDINT
VAR_INPUT
	Run						: UINT;
	ptArray					: POINTER TO ARRAY[0..MATHOLES_COUNT] OF ST_Coordinate;
END_VAR

VAR
	tmpCount				: UDINT;
	tmpDest					: POINTER TO ARRAY[0..MATHOLES_COUNT] OF ST_Coordinate;
	ni						: UINT;
END_VAR
IF ptArray = 0 THEN
	RETURN;
END_IF

MEMSet(ptArray,0,SIZEOF(POINTER TO ARRAY[0..MATHOLES_COUNT] OF ST_Coordinate));

/// DEFINE VARIABLES, CHECK REFERENZES
//IF NOT __ISVALIDREF(refMat) THEN	RETURN;	END_IF 

HolesOfRun := tmpCount := Count_HolesOfRun(Run);
IF tmpCount <= 0 OR tmpCount > MATHOLES_COUNT THEN	RETURN;	END_IF

/// COPY ELEMENTS IN ARRAY
tmpCount := 0;
tmpDest := ptArray;

FOR ni := 0 TO MATELEMENTS_COUNT DO
	tmpCount := HolesOfElement(Run, ni, tmpDest);
	tmpDest := tmpDest + SIZEOF(ST_Coordinate)*tmpCount;
END_FOR
END_METHOD

METHOD LoadMat
VAR_IN_OUT
	Mat						: ST_Mat;
END_VAR
nRunNr:= 0;
MEMSET(ADR(stCoordinates), 0, SIZEOF(stCoordinates));
eCoordinatesSortState := E_CoordinatesSortState.eCoordinatesSortState_undefined;
stMat := Mat;
nCorrdinatesCount := 0;
END_METHOD

PROPERTY Mat : REFERENCE TO ST_Mat
GET
Mat REF= stMat;
END_GET
SET
stMat := Mat;
END_SET
END_PROPERTY

PROPERTY MaxDistanceX : LREAL
GET
VAR
	ni				: UDINT;
	tmpDistance		: LREAL;
END_VAR
IF eCoordinatesSortState <> E_CoordinatesSortState.eCoordinatesSortState_resorted_v1 THEN
	MaxDistanceX := 0;
	RETURN;
END_IF

tmpDistance := 0;

FOR ni:= 0 TO nCorrdinatesCount-2 DO
	tmpDistance := MAX(tmpDistance, ABS(stCoordinates[ni].fX - stCoordinates[ni+1].fX));
END_FOR

MaxDistanceX := tmpDistance;
END_GET
END_PROPERTY

PROPERTY MaxDistanceY : LREAL
GET
VAR
	ni				: UDINT;
	tmpDistance		: LREAL;
END_VAR
IF eCoordinatesSortState <> E_CoordinatesSortState.eCoordinatesSortState_resorted_v1 THEN
	MaxDistanceY := 0;
	RETURN;
END_IF

tmpDistance := 0;

FOR ni:= 0 TO nCorrdinatesCount-2 DO
	tmpDistance := MAX(tmpDistance, ABS(stCoordinates[ni].fY - stCoordinates[ni+1].fY));
END_FOR

MaxDistanceY := tmpDistance;
END_GET
END_PROPERTY

/// Reset component logic
{attribute 'object_name' := 'Reset'}
METHOD Reset
// base logic run
SUPER^.Reset();

nRunNr:= 0;
MEMSET(ADR(stCoordinates), 0, SIZEOF(stCoordinates));
eCoordinatesSortState := E_CoordinatesSortState.eCoordinatesSortState_undefined;
nCorrdinatesCount := 0;
END_METHOD

METHOD ResortCoordinates : E_OperationResult
VAR_INPUT
	ResortVersion		 	: E_CoordinatesSortState;
END_VAR

VAR
	fTmpX					: REAL;
	
	bResort					: BOOL;
	nStartIdx				: UDINT;
	nEndIdx					: UDINT;
	
	ni, nj					: UDINT;
END_VAR

VAR_INST	
	tmp						: ST_Coordinate;
END_VAR
ResortCoordinates := E_OperationResult.eOperationResult_NOk;
IF nCorrdinatesCount <= 0 THEN
	RETURN;
END_IF

fTmpX := stCoordinates[0].fX;
nStartIdx := 0;
bResort := FALSE;
nEndIdx := 0;

FOR ni:= 0 TO nCorrdinatesCount-1 DO

	IF ni = nCorrdinatesCount-1 THEN	// letzte Element
		nEndIdx := ni;			
	ELSIF fTmpX = stCoordinates[ni].fX THEN
		CONTINUE;	
	ELSE
		nEndIdx := ni-1;	
	END_IF
	
	IF bResort THEN	
		FOR nj:= 0 TO ((nEndIdx-nStartIdx)/2) DO
			tmp := stCoordinates[nEndIdx - nj];
			stCoordinates[nEndIdx - nj] := stCoordinates[nStartIdx + nj];
			stCoordinates[nStartIdx + nj] := tmp;	
		END_FOR	
		bResort := FALSE;
	ELSE
		bResort := TRUE;	
	END_IF
	
	fTmpX := stCoordinates[ni].fX;
	nStartIdx := ni;

END_FOR

ResortCoordinates := E_OperationResult.eOperationResult_Ok;
eCoordinatesSortState := E_CoordinatesSortState.eCoordinatesSortState_resorted_v1;
END_METHOD

/// Run component logic
{attribute 'object_name' := 'Run'}
METHOD Run : E_ComponentState
// base logic run
Run := SUPER^.Run();
END_METHOD

METHOD SortRun : E_OperationResult
VAR_INPUT
	Run						: UINT;
END_VAR
VAR
	stack_count: UINT;					(* Laufvariable Stack*)
	stack: ARRAY[1..4096] OF UDINT;		(* Stackgröße~ 1,6*Log(n)/log(2) *)
										(* Stackgröße 32 => ~1 Mio Elemente *)
										(* Stackgröße auf 64 erhöht da sortierfehler aufgetreten sind *)
	links: UDINT;						(* Anfangselement des Arrays *)
	rechts: UDINT;						(* Endelement des Arrays *)
	
	i: UDINT;							(* Laufvariable1 *)
	j: UDINT;							(* Laufvariable2 *)
	ende_innen: BOOL;					(* Ende innere Schleife *)
	ende_aussen: BOOL;					(* Ende äußere Schleife *)
	
END_VAR
VAR_INST
	pivot					: ST_Coordinate;				(* temporärer Schwellwert für Tauschbedingung *)
	tmp						: ST_Coordinate;
END_VAR
SortRun := E_OperationResult.eOperationResult_NOk;

SortRun := ConvertRun(Run);
(* Startwerte zur Arraygröße *)
links := 1;						(* Anfangselement des Arrays *)
rechts := nCorrdinatesCount;//SHR(size,2);		(* Endelement des Arrays *)
stack_count := 1;//1;			(* Laufvariable Stack *)

WHILE NOT ende_aussen DO						(* äußere Schleife *)
	IF links < rechts THEN
		pivot := stCoordinates[SHR(rechts+links,1)-1];			(* Wert des mittleren Elements als Pivot-Wert *)
		i := links -1;
		j := rechts +1;
		
		(* innere Schleife, teile Feld *)
		ende_innen := FALSE;
		REPEAT

			(* steigende Reihenfolge *)
			REPEAT	i := i+1;	UNTIL (Cmp_Coordinates(ADR(stCoordinates[i-1]), ADR(pivot)) >= 0) OR NOT (i < rechts)	END_REPEAT;
			REPEAT	j := j-1;	UNTIL (Cmp_Coordinates(ADR(stCoordinates[j-1]), ADR(pivot)) <= 0) OR NOT (j > links)	END_REPEAT;
			
			IF i >= j THEN
				ende_innen := TRUE;
			ELSE
				tmp := stCoordinates[j-1];
				stCoordinates[j-1] := stCoordinates[i-1];
				stCoordinates[i-1] := tmp;	
			END_IF;

		UNTIL ende_innen END_REPEAT;
		

		(* Push stack *)
		stack[stack_count] := rechts;		(* rechten Teil später sortieren *)
		IF Stack_count < 4096 THEN
			stack_count := stack_count +1;
		ELSE
			ende_aussen := TRUE;
			SortRun := E_OperationResult.eOperationResult_NOk;
		END_IF;

		(* linken Teil sortiern *)
		rechts := MAX(links, i-1);

	ELSE

		IF stack_count = 1 THEN
			ende_aussen := TRUE;
		ELSE

			links := rechts+1;

			(* pop stack *)
			stack_count := stack_count -1;		(* jetzt rechten Teil sortierne *)
			rechts:= stack[stack_count];
		END_IF;

	END_IF;

END_WHILE;

eCoordinatesSortState := E_CoordinatesSortState.eCoordinatesSortState_sorted;
SortRun := E_OperationResult.eOperationResult_Ok;
END_METHOD

END_FUNCTION_BLOCK

// ---- Components/PunchEngine/FB_PunchEngine.TcPOU
FUNCTION_BLOCK FB_PunchEngine EXTENDS FB_ComponentBase

VAR PERSISTENT
	nPunchCount					: UDINT;
	fZeroOffset					: LREAL;
END_VAR

VAR	

	// Sequencer
	fbSeq						: FB_Sequence;
	fbSeqOutletBelt				: FB_Sequence;
	
	fVelocity					: LREAL;
	fAcceleration				: LREAL;
	
	fMovePosition				: LREAL;
	bJogPos						: BOOL;
	bJogNeg						: BOOL;
	nPunchRemain				: UINT;
	
	bEnableOutletBelt			: BOOL;
	tIntervallOutletbelt		: TIME;
	tOutletbeltRuntime			: TIME;

	// Watch Variables
	bOutsideMat					: BOOL;
	bPunchDone					: BOOL;
	refObstacle					: REFERENCE TO BOOL;	
	fTravelPosition				: LREAL;
		
	// Parameter
	fPunchHeight				: REAL;
	fPunchHeightAddon			: REAL := 3;
	fPunchVelocity				: LREAL;
	fPunchAcceleration			: LREAL;
	
	// Settings	
	fRodLenght					: REAL;
	fCrankThrow					: REAL;
		
	fMaxVelocity				: LREAL;
	fMinVelocity				: LREAL;
	fDefaultVelocity			: LREAL;
	
	fMaxAcceleration			: LREAL;
	fMinAcceleration			: LREAL;
	fDefaultAcceleration		: LREAL;
	
	fToleranceWindowMM			: LREAL := 0.5;
	fToleranceWindowDeg			: LREAL := 5;
	
	// TorquwLimit
	nTorqueLimit				: INT := 100;
	nTorqueLimitPos				: INT := 100;
	nTorqueLimitNeg				: INT := 10;
		
	// Axis
	bEnable						: BOOL := TRUE;
	refEnable					: REFERENCE TO BOOL;
	fbPunchAxis					: FB_AxisDriver;
	fbOutletbelt				: FB_DigitalOutput;


END_VAR

//TODO: abtransportband!!!!!!

METHOD _Halt : BOOL
VAR_INPUT
END_VAR
fbSeq.Name := 'Halt';

CASE fbSeq.Step OF
	

0	 :	fbSeq.StepDefinition('Punchaxis Halt', T#0S);

		fbPunchAxis.posTorqueLimit := nTorqueLimit;
		fbPunchAxis.negTorqueLimit := nTorqueLimit;
		fbPunchAxis.Halt();		
		fbSeq.NextStep(10);
	
		
10	 :	fbSeq.StepDefinition('', T#0S);
		IF fbPunchAxis.NotMoving THEN
			fbSeq.Finish();
		END_IF
			
END_CASE
END_METHOD

METHOD _Home : BOOL
VAR_INPUT
END_VAR
fbSeq.Name := 'Home';

CASE fbSeq.Step OF
	

0	 :	fbSeq.StepDefinition('Reset Axis', T#0S);

		fbSeq.NextStep(10);
	
	
10	 :	fbSeq.StepDefinition('Set Zero-Position', T#0S);

		fbSeq.NextStep(20);	

		
20	 :	fbSeq.StepDefinition('Move to Zero Postion', T#0S);

		fbSeq.NextStep(30);	

		
30	 :	fbSeq.StepDefinition('', T#0S);

		fbSeq.NextStep(40);

		
40	 :	fbSeq.StepDefinition('', T#0S);

		fbSeq.NextStep(50);

		
50	 :	fbSeq.StepDefinition('', T#0S);

		fbSeq.Finish();

END_CASE
END_METHOD

METHOD _Jog : BOOL
VAR_INPUT
END_VAR
fbSeq.Name := 'Jog';

CASE fbSeq.Step OF
	

0	 :	fbSeq.StepDefinition('Halt Axis', T#0S);
		fbPunchAxis.posTorqueLimit := nTorqueLimit;
		fbPunchAxis.negTorqueLimit := nTorqueLimit;
		fbPunchAxis.Halt();
		fbSeq.NextStep(10);
	
10	 :	fbSeq.StepDefinition('Jog Axis', T#0S);
	
		IF bJogPos OR bJogNeg THEN
			fbPunchAxis.JogAcc(bJogPos , bJogNeg);
		ELSE
			fbSeq.NextStep(20);
		END_IF		
		
20	 :	fbSeq.StepDefinition('Jog Finish', T#0S);
		fbSeq.Finish();

END_CASE
END_METHOD

METHOD _Move : BOOL
VAR
	stMovModParameter			: ST_AxisMoveModParameter;
END_VAR
fbSeq.Name := 'Move';

CASE fbSeq.Step OF
	

0	 :	fbSeq.StepDefinition('Calculate nearest Position', T#0S);
		fbPunchAxis.posTorqueLimit := nTorqueLimit;
		fbPunchAxis.negTorqueLimit := nTorqueLimit;
		
		IF CrankAngle >= 180 THEN
			stMovModParameter.eDirection := MC_Direction.MC_Positive_Direction;
		ELSIF CrankAngle < 180 THEN
			stMovModParameter.eDirection := MC_Direction.MC_Shortest_Way;
		END_IF
		
		stMovModParameter.fPosition := PistonTravelToDeg1(fMovePosition);
		stMovModParameter.fVelocity := fVelocity;
		stMovModParameter.fAcceleration := fAcceleration;
		fbPunchAxis.MoveModEx(stMovModParameter);	
		fbSeq.NextStep(10);
	
	
10	 :	fbSeq.StepDefinition('Position reached', T#0S);
		IF fbPunchAxis.TargetReachedMod(fToleranceWindowDeg) THEN
			fbSeq.Finish();
		END_IF

		
END_CASE
END_METHOD

METHOD _OutletBelt : BOOL
VAR_INPUT
END_VAR
CASE fbSeqOutletBelt.Step OF
	
	0	:	fbSeqOutletBelt.StepDefinition('OutletBelt waiting', T#0S);
			fbSeqOutletBelt.NextStepTransition(10, bEnableOutletBelt);
	
	10	:	fbOutletbelt.SwitchState(TRUE);
			fbSeqOutletBelt.NextStep(20);
			
	20	:	fbSeqOutletBelt.StepDefinition('OutletBelt running', T#0S);
			fbSeqOutletBelt.NextStepDelay(tOutletbeltRuntime, 30);
	
	30	:   fbOutletbelt.SwitchState(FALSE);
			bEnableOutletBelt := FALSE;
			fbSeqOutletBelt.NextStep(40);

	40	:	fbSeqOutletBelt.StepDefinition('OutletBelt resting', T#0S);
			fbSeqOutletBelt.NextStepDelay(tintervallOutletbelt, 0);
	

END_CASE
END_METHOD

METHOD _Punch : BOOL
VAR
	stMovModParameter			: ST_AxisMoveModParameter;
	stMovAddParameter			: ST_AxisMoveAddParameter;
	fPosition					: REAL;
END_VAR
fbSeq.Name := 'Punch';

CASE fbSeq.Step OF
	
0	 :	fbSeq.StepDefinition('Move To Start-Point', T#0S);
		IF fbPunchAxis.TargetReachedMod(fToleranceWindowDeg) THEN
			fbSeq.NextStep(20);
			RETURN;
		END_IF
		
		IF CrankAngle >= 180 THEN
			stMovModParameter.eDirection := MC_Direction.MC_Positive_Direction;
		ELSIF CrankAngle < 180 THEN
			stMovModParameter.eDirection := MC_Direction.MC_Shortest_Way;
		END_IF
		
		fbPunchAxis.posTorqueLimit := nTorqueLimit;
		fbPunchAxis.negTorqueLimit := nTorqueLimit;
				
		stMovModParameter.fPosition := 0;
		stMovModParameter.fVelocity := fDefaultVelocity;
		stMovModParameter.fAcceleration := fDefaultAcceleration;
		stMovModParameter.eBufferMode := MC_BufferMode.MC_Aborting;
		fbPunchAxis.MoveModEx(stMovModParameter);	
		fbSeq.NextStep(10);	
	
10	 :	fbSeq.StepDefinition('Start-Point reached', T#0S);
		IF fbPunchAxis.TargetReachedMod(fToleranceWindowDeg) THEN
			fbSeq.NextStep(20);
		END_IF

20	 :	fbSeq.StepDefinition('Start Punch', T#0S);	
		
		fbPunchAxis.posTorqueLimit := nTorqueLimitPos;
		fbPunchAxis.negTorqueLimit := nTorqueLimitNeg;

		stMovAddParameter.fDistance := 360;
		stMovAddParameter.fVelocity := fPunchVelocity;
		stMovAddParameter.fAcceleration := fPunchAcceleration;
		stMovAddParameter.eBufferMode := MC_BufferMode.MC_Aborting;
		fbPunchAxis.MoveAddEx(stMovAddParameter);	
		fbSeq.NextStep(30);	
		
30	 :	fbSeq.StepDefinition('Punching', T#0S);
		IF InsideMat THEN
			fbSeq.NextStep(40);	
		END_IF			
		
40	 :	fbSeq.StepDefinition('Punching done', T#0S);
		IF OutsideMat THEN
			bPunchDone := TRUE;
			nPunchRemain := nPunchRemain - 1;
			nPunchCount := nPunchCount + 1;
			fbSeq.NextStep(50);	
		END_IF			

50   :	fbSeq.StepDefinition('Check for Continue Punching', T#0S);  
		IF nPunchRemain > 0 THEN
			fbSeq.NextStep(20);	
			RETURN;
		END_IF
		
		fbPunchAxis.posTorqueLimit := nTorqueLimit;
		fbPunchAxis.negTorqueLimit := nTorqueLimit;
			
		IF NOT fbPunchAxis.Moving THEN
			fbSeq.Finish();			
		END_IF	
END_CASE
END_METHOD

/// Actual amplifier temp. [°C]
PROPERTY AmplifierTemp : LREAL
GET
/// Actual amplifier temp. [°C]
AmplifierTemp := fbPunchAxis.AmplifierTemp;
END_GET
END_PROPERTY

PROPERTY BDC : BOOL
GET
BDC := ABS(CrankAngle-180) < fToleranceWindowDeg;
END_GET
END_PROPERTY

PROPERTY CrankAngle : LREAL
GET
VAR
	refAxis				: REFERENCE TO AXIS_REF;
END_VAR
CrankAngle := fbPunchAxis.ActModuloPos;
END_GET
END_PROPERTY

METHOD DegToPistonTravel : LREAL
VAR_INPUT
	fAngle						: LREAL;
END_VAR
VAR
	a							: LREAL;
	b							: LREAL;
	h							: LREAL;
END_VAR
a := fCrankThrow * SIN (DEG_TO_RAD(fAngle));
b := fCrankThrow * COS (DEG_TO_RAD(fAngle));
IF fRodLenght*fRodLenght-a*a < 0 THEN
	RETURN;
END_IF

h := SQRT(fRodLenght*fRodLenght-a*a);

DegToPistonTravel := fCrankThrow - fRodLenght + h - b;


// MANFRED
//a := fCrankThrow * SIN (DEG_TO_RAD(fAngle));
//b := fCrankThrow * COS (DEG_TO_RAD(fAngle));
//
//h1 := fCrankThrow - b;
//h2 := SQRT(fRodLenght*fRodLenght-a*a);
//
//DegToPistonTravel := 2 * fCrankThrow + fRodLenght - h1 - h2;



/// http://www.3d-meier.de/tut16/Kurbel1/Seite1.html	
//DegToPistonTravel := fRodLenght + fCrankThrow - (fCrankThrow * COS(DEG_TO_RAD(fAngle)) + fRodLenght * SQRT(1 - SQRT(fCrankThrow/fRodLenght) * SQRT(SIN(DEG_TO_RAD(fAngle)))));
END_METHOD

METHOD FB_init : BOOL
VAR_INPUT
	bInitRetains : BOOL; // if TRUE, the retain variables are initialized (warm start / cold start)
	bInCopyCode : BOOL;  // if TRUE, the instance afterwards gets moved into the copy code (online change)
END_VAR
eTyp := E_ComponentType.eComponentType_PunchEngine;
END_METHOD

METHOD Halt : E_OperationResult
VAR_INPUT
END_VAR
// init result pessimistic
Halt := E_OperationResult.eOperationResult_NOk;

fbSeq.Start(E_PunchEngineCmd.cmdHalt);

Halt := E_OperationResult.eOperationResult_Ok;
END_METHOD

METHOD Home : E_OperationResult
VAR_INPUT
END_VAR
// init result pessimistic
Home := E_OperationResult.eOperationResult_NOk;

fbSeq.Start(E_PunchEngineCmd.cmdHome);

Home := E_OperationResult.eOperationResult_Ok;
END_METHOD

PROPERTY Homed : BOOL
GET
Homed := fbPunchAxis.Homed;
END_GET
END_PROPERTY

PROPERTY Homing : BOOL
GET
Homing := fbPunchAxis.Homing;
END_GET
END_PROPERTY

PROPERTY InsideMat : BOOL
GET
InsideMat := NOT bOutsideMat;
END_GET
END_PROPERTY

METHOD Jog : E_OperationResult
VAR_INPUT
	JogPos					: BOOL;
	JogNeg					: BOOL;
END_VAR
// init result pessimistic
Jog := E_OperationResult.eOperationResult_NOk;

IF fbSeq.SequenceId <> E_PunchEngineCmd.cmdJog THEN
	fbSeq.Start(E_PunchEngineCmd.cmdJog);
//	RETURN;
END_IF

IF JogPos AND JogNeg THEN
	RETURN;
END_IF

bJogPos := JogPos;
bJogNeg := JogNeg;

Jog := E_OperationResult.eOperationResult_Ok;
END_METHOD

METHOD JogStop : E_OperationResult
// init result pessimistic
JogStop := E_OperationResult.eOperationResult_NOk;

bJogPos := FALSE;
bJogNeg := FALSE;

JogStop := E_OperationResult.eOperationResult_Ok;
END_METHOD

/// Actual motor temp. [°C]
PROPERTY MotorTemp : LREAL
GET
/// Actual motor temp. [°C]
MotorTemp := fbPunchAxis.MotorTemp;
END_GET
END_PROPERTY

METHOD MoveBDC : E_OperationResult
VAR_INPUT
END_VAR
// init result pessimistic
MoveBDC := E_OperationResult.eOperationResult_NOk;

IF ABS(CrankAngle-180) < fToleranceWindowDeg THEN
	RETURN;
END_IF

fMovePosition := 2*fCrankThrow;
fVelocity := fDefaultVelocity; //MAX(MIN(fMaxVelocity, Velocity),fMinVelocity);	
fAcceleration := fDefaultAcceleration;
fbSeq.Start(E_PunchEngineCmd.cmdMove);

MoveBDC := E_OperationResult.eOperationResult_Ok;
END_METHOD

METHOD MovePos : E_OperationResult
VAR_INPUT
	MovePosition			: LREAL;
	Velocity				: LREAL;
END_VAR
// init result pessimistic
MovePos := E_OperationResult.eOperationResult_NOk;

IF ABS(DegToPistonTravel(CrankAngle)-MovePosition) < fToleranceWindowMM THEN
	RETURN;
END_IF

fMovePosition := MovePosition;
fVelocity := MAX(MIN(fMaxVelocity, Velocity),fMinVelocity);	
fAcceleration := fDefaultAcceleration;
fbSeq.Start(E_PunchEngineCmd.cmdMove);

MovePos := E_OperationResult.eOperationResult_Ok;
END_METHOD

METHOD MoveSTART : E_OperationResult
VAR_INPUT
END_VAR
// init result pessimistic
MoveSTART := E_OperationResult.eOperationResult_NOk;

fMovePosition := fCrankThrow*2 - fPunchHeight - fPunchHeightAddon ;
fVelocity := fDefaultVelocity; //MAX(MIN(fMaxVelocity, Velocity),fMinVelocity);	
fAcceleration := fDefaultAcceleration;
fbSeq.Start(E_PunchEngineCmd.cmdMove);

MoveSTART := E_OperationResult.eOperationResult_Ok;
END_METHOD

METHOD MoveTDC : E_OperationResult
VAR_INPUT
END_VAR
// init result pessimistic
MoveTDC := E_OperationResult.eOperationResult_NOk;

IF TDC THEN
	RETURN;
END_IF

fMovePosition := 0;
fVelocity := fDefaultVelocity; //MAX(MIN(fMaxVelocity, Velocity),fMinVelocity);	
fAcceleration := fDefaultAcceleration;
fbSeq.Start(E_PunchEngineCmd.cmdMove);

MoveTDC := E_OperationResult.eOperationResult_Ok;
END_METHOD

PROPERTY Moving : BOOL
GET
Moving := fbPunchAxis.Moving;
END_GET
END_PROPERTY

PROPERTY NotMoving : BOOL
GET
NotMoving := fbPunchAxis.NotMoving;
END_GET
END_PROPERTY

METHOD OutletBeltJog : BOOL
VAR_INPUT
	Enable					: BOOL;
END_VAR
//bEnableOutletBelt := FALSE;
//fbSeqOutletBelt.Init();
IF bEnableOutletBelt THEN
	RETURN;
END_IF
fbOutletbelt.SwitchState(Enable);
END_METHOD

METHOD OutletBeltOnce : BOOL
VAR_INPUT
END_VAR
fbSeqOutletBelt.Init();
tintervallOutletbelt := T#0S;
bEnableOutletBelt := TRUE;
END_METHOD

METHOD OutletBeltSeq : BOOL
VAR_INPUT
	bEnable				: BOOL;
	tIntervall			: UINT;
END_VAR
IF NOT bEnable THEN
	bEnableOutletBelt := FALSE;
	fbSeqOutletBelt.Init();
	fbOutletbelt.SwitchState(FALSE);
ELSE
	bEnableOutletBelt := bEnable;
	tIntervallOutletbelt := DINT_TO_TIME(1000*UINT_TO_DINT(tIntervall));
END_IF
END_METHOD

PROPERTY OutsideMat : BOOL
GET
OutsideMat := bOutsideMat;
END_GET
END_PROPERTY

PROPERTY Override : LREAL
GET
Override := fbPunchAxis.Override;
END_GET
SET
IF Override <> fbPunchAxis.Override THEN
	fbPunchAxis.Override := Override;
	fbPunchAxis.posTorqueLimit := 100;
	fbPunchAxis.negTorqueLimit := 100;
END_IF
END_SET
END_PROPERTY

METHOD PistonTravelToDeg1 : LREAL
VAR_INPUT
	fPistonTravel		: LREAL;
END_VAR
VAR
	h					: LREAL;
	tmp					: LREAL;
END_VAR
IF fPistonTravel > 2 * fCrankThrow OR fPistonTravel < 0 THEN
	RETURN;
END_IF

IF fPistonTravel = 0 THEN
	PistonTravelToDeg1:= 0;	
	RETURN;
END_IF

IF fPistonTravel = 2 * fCrankThrow THEN
	PistonTravelToDeg1:= 180;	
	RETURN;
END_IF

h := fPistonTravel + fRodLenght - fCrankThrow;

tmp := (-fRodLenght*fRodLenght + h*h + fCrankThrow*fCrankThrow)/(2*h*fCrankThrow);

PistonTravelToDeg1:= 180 - rad_to_deg(ACOS(tmp));
END_METHOD

METHOD PistonTravelToDeg2 : LREAL
VAR_INPUT
	fPistonTravel		: LREAL;
END_VAR
VAR
	h					: LREAL;
	tmp					: LREAL;
END_VAR
IF fPistonTravel > 2 * fCrankThrow OR fPistonTravel < 0 THEN
	RETURN;
END_IF

IF fPistonTravel = 0 THEN
	PistonTravelToDeg2:= 0;	
	RETURN;
END_IF

IF fPistonTravel = 2 * fCrankThrow THEN
	PistonTravelToDeg2:= 180;	
	RETURN;
END_IF

h := fPistonTravel + fRodLenght - fCrankThrow;

tmp := (-fRodLenght*fRodLenght + h*h + fCrankThrow*fCrankThrow)/(2*h*fCrankThrow);

PistonTravelToDeg2:= 180 + rad_to_deg(ACOS(tmp));
END_METHOD

METHOD Punch : E_OperationResult
VAR_INPUT
	Continuous				: BOOL;
END_VAR

VAR
	stMovAddParameter			: ST_AxisMoveAddParameter;
END_VAR
// init result pessimistic
Punch := E_OperationResult.eOperationResult_NOk;

fVelocity := MAX(MIN(fMaxVelocity, fPunchVelocity),fMinVelocity);	
fAcceleration := MAX(MIN(fMaxAcceleration, fAcceleration),fMinAcceleration);

bPunchDone:= FALSE;

IF fbseq.SequenceId <> E_PunchEngineCmd.cmdPunch THEN
	nPunchRemain := 1;
	fbSeq.Start(E_PunchEngineCmd.cmdPunch);	
END_IF

IF Continuous THEN
	nPunchRemain := nPunchRemain + 1;
END_IF

Punch := E_OperationResult.eOperationResult_Ok;
END_METHOD

PROPERTY PunchCount : UDINT
GET
PunchCount := nPunchCount;
END_GET
END_PROPERTY

PROPERTY PunchDone : BOOL
GET
PunchDone := bPunchDone;
END_GET
END_PROPERTY

PROPERTY PunchHeight : REAL
GET
PunchHeight := fPunchHeight;
END_GET
SET
fPunchHeight := PunchHeight;
END_SET
END_PROPERTY

PROPERTY Punching : BOOL
GET
Punching := fbSeq.SequenceId = E_PunchEngineCmd.cmdPunch AND fbSeq.State = E_SequenceState.eSequenceState_running;
END_GET
END_PROPERTY

PROPERTY Ready : BOOL
GET
Ready := fbPunchAxis.MotionState <> MC_AXISSTATE_DISABLED;
END_GET
END_PROPERTY

/// Reset component logic
{attribute 'object_name' := 'Reset'}
METHOD Reset
// base logic run
SUPER^.Reset();

fbPunchAxis.Reset();
fbPunchAxis.TorqueLimit := 100;
fbPunchAxis.posTorqueLimit := 100;
fbPunchAxis.negTorqueLimit := 100;

fbOutletbelt.Reset();
nPunchRemain := 0;

fbSeq.Init();			
fbSeqOutletBelt.Init();
END_METHOD

/// Run component logic
{attribute 'object_name' := 'Run'}
METHOD Run : E_ComponentState
// run Base Logic
Run := SUPER^.Run();

IF __ISVALIDREF(refEnable) THEN
	bEnable := refEnable;
END_IF

// run Axis Driver
fbPunchAxis.Run();
fbPunchAxis.Enable := bEnable;
fbPunchAxis.EnablePos := bEnable;
fbPunchAxis.EnableNeg := bEnable;


fbOutletbelt.Run();

// watch Position
fTravelPosition := DegToPistonTravel(CrankAngle);
bOutsideMat := DegToPistonTravel(CrankAngle) < (fCrankThrow*2 - fPunchHeight - fPunchHeightAddon);  

// run Sequences
fbSeq.Enable := TRUE;
fbSeq.Base(FALSE, FALSE);
CASE fbSeq.SequenceId OF	
	E_PunchEngineCmd.cmdMove:	_Move();
	E_PunchEngineCmd.cmdHalt:	_Halt();	
	E_PunchEngineCmd.cmdPunch:	_Punch();	
	E_PunchEngineCmd.cmdHome:	_Home();
	E_PunchEngineCmd.cmdJog:	_Jog();
END_CASE

fbSeqOutletBelt.Enable := TRUE;
fbSeqOutletBelt.Base(FALSE, FALSE);				
_OutletBelt();
END_METHOD

METHOD SetObstacle : BOOL
VAR_IN_OUT
	Obstacle			: BOOL;
END_VAR
refObstacle REF= Obstacle;
END_METHOD

METHOD Setup
VAR_INPUT
	eAxis					: E_Axis;
	eDigitalOutlet			: E_DigitalOutput;
END_VAR
fbPunchAxis.Name := 'Punch Axis';
fbPunchAxis.SetAxisReference(COMP.astAxisRef[eAxis_Punch], COMP.astAxisIO[eAxis_Punch].stIn, COMP.astAxisIO[eAxis_Punch].stOut);
fbPunchAxis.AxisType := E_AxisType.AX5xxx;
fbPunchAxis.DefaultParameter.stMovAbsPrm.fVelocity := 30;
fbPunchAxis.Active := TRUE;
fbPunchAxis.Override := 100;
fbPunchAxis.DefaultParameter.stJogAccPrm.fFastSpeed := 20;
fbPunchAxis.DefaultParameter.stJogAccPrm.fSlowSpeed := 1;
fbPunchAxis.DefaultParameter.stJogAccPrm.tAccTime := T#5S;
fbPunchAxis.EnableLimitSensor:= FALSE;	


fbOutletbelt.Name := 'Outletbelt';
fbOutletbelt.SetReferences(COMP.aStDigitalOutputIO[eDigitalOutput_OutletBelt]);
fbOutletbelt.Active := TRUE;
tOutletbeltRuntime := T#25S;


fMaxVelocity		 := 1111;
fMinVelocity		 := 10;
fDefaultVelocity	 := 180;

fMaxAcceleration	 := 1000000;
fMinAcceleration	 := 0;
fDefaultAcceleration := 0;

fToleranceWindowMM	 := 0.5;
fToleranceWindowDeg	 := 1.5;
END_METHOD

METHOD SetupCrank : BOOL
VAR_INPUT
	fRodLenght				: REAL;
	fCrankThrow				: REAL;
END_VAR
THIS^.fRodLenght	:= fRodLenght;
THIS^.fCrankThrow	:= fCrankThrow;
END_METHOD

METHOD SetupEnable : BOOL

VAR_IN_OUT
	bEnable					: BOOL;
END_VAR
refEnable REF= bEnable;
END_METHOD

METHOD SetupPunch : BOOL
VAR_INPUT
	PunchHeight					: REAL;
	PunchHeightAddon			: REAL;
	MaxVelocity					: LREAL;
	MaxAcceleration				: LREAL;
	TimeBetweenPunch			: LREAL;
END_VAR

VAR
	tmpAngle					: LREAL;
END_VAR
IF TimeBetweenPunch = 0  THEN
	fPunchVelocity := MaxVelocity;
	fPunchAcceleration := MaxAcceleration;
	RETURN;
END_IF

fPunchHeight := PunchHeight;  
fPunchHeightAddon := PunchHeightAddon;


tmpAngle := PistonTravelToDeg1(fCrankThrow*2 - PunchHeight - PunchHeightAddon);

fPunchVelocity := MIN((2*tmpAngle/TimeBetweenPunch), MaxVelocity);
fPunchAcceleration := MaxAcceleration;
END_METHOD

METHOD SetZeroOffset
VAR
	stParam				: st_AxisHomingParameter;
	
END_VAR
fZeroOffset := fbPunchAxis.ActModuloPos;

stParam.fPosition:= 0;
stParam.eHomingMode := MC_HomingMode.MC_Direct; 

fbPunchAxis.HomeEx(stParam);
END_METHOD

PROPERTY TargetReached : BOOL
GET
TargetReached := fbPunchAxis.TargetReachedMod(fToleranceWindowDeg);
END_GET
END_PROPERTY

PROPERTY TDC : BOOL
GET
TDC := ABS(CrankAngle) < fToleranceWindowDeg;
END_GET
END_PROPERTY

/// Actual torque [Nm]
PROPERTY Torque : LREAL
GET
/// Actual torque [Nm]
Torque := fbPunchAxis.Torque;
END_GET
END_PROPERTY

/// The torque limit for both directions. [Nm]
PROPERTY TorqueLimit : INT
GET
/// The torque limit for both directions. [1/10%]
TorqueLimit := nTorqueLimit;
END_GET
SET
nTorqueLimit := TorqueLimit;
END_SET
END_PROPERTY

/// The torque limit for both directions. [Nm]
PROPERTY TorqueLimitNeg : INT
GET
/// The torque limit for both directions. [1/10%]
TorqueLimitNeg := nTorqueLimitNeg;
END_GET
SET
nTorqueLimitNeg := TorqueLimitNeg;
END_SET
END_PROPERTY

/// The torque limit for both directions. [Nm]
PROPERTY TorqueLimitPos : INT
GET
/// The torque limit for both directions. [1/10%]
TorqueLimitPos := nTorqueLimitPos;
END_GET
SET
nTorqueLimitPos := TorqueLimitPos;
END_SET
END_PROPERTY

PROPERTY Velocity : LREAL
GET
Velocity := fVelocity;
END_GET
END_PROPERTY

PROPERTY ZeroOffset : LREAL
GET
ZeroOffset := fZeroOffset;
END_GET
END_PROPERTY

END_FUNCTION_BLOCK

// ---- BaseComponents/AxisDriver/FB_AxisDriver.TcPOU
/// Axis driver function block
FUNCTION_BLOCK FB_AxisDriver EXTENDS FB_ComponentBase IMPLEMENTS ITFMotionComponent
VAR_INPUT
	/// AmsNetId of the IPC 
	IPCNetID: T_AmsNetId := '';
END_VAR
VAR_OUTPUT
	/// Fehlerzustand
	Error: BOOL;
	/// Position der Achse
	Position: LREAL;
	/// Aktuelle Positionen mit gelatchten Objektposition gleich
	bLatchedObjPositionOK					:BOOL;
END_VAR
VAR
	/// private workflow var`s
	/// component type
	bEnable: BOOL;
	bEnableLimit: BOOL := FALSE;
	bEnablePos: BOOL;
	bEnableNeg: BOOL;
	
	nLimitPos		: LREAL;
	nLimitNeg		: LREAL;
	
	fPositionBias	: LREAL;
	fFeedConstant	: LREAL;
	
	
	bSafetyCardAct: BOOL;
	eMasterAxisId: E_Axis;
	eAxisType: E_AxisType;
	stDefaultPrm: ST_AxisDriverParameter;
	ptDefaultPrm: POINTER TO ST_AxisDriverParameter;
	nErrorID: UDINT;
	bErrDiagActive: BOOL;
	sMsg: T_MaxString;
	/// requested motion command
	eCommandRequest: E_MotionCommand;
	fPosRequest	: LREAL;
	fPosLatched	: LREAL;
	/// actual motion command
	eCommandExecute: E_MotionCommand;
	
	/// Axis ID and reference
	eAxisId: E_Axis;
	fbAxisRef: REFERENCE TO AXIS_REF;
	/// Additional (direct) linked inputs
	stIn: REFERENCE TO ST_AxisIn;
	/// Additional (direct) linked outputs
	stOut: REFERENCE TO ST_AxisOut;
	/// Device ref: contains sNetID of EcMaster, nSlaveAddr of EcDrive, nDriveNo of EcDrive, either preset or read from NC 
	stDriveRef: ST_DriveRef;
	///	AX5000 - axes diag + reset 
	fbAX5xxxDiag: FB_AX5000Diag;
	stAX5xxxDiag: ST_AX5000Diag;
	
	/// FB for axis enabling
	fbPower: MC_Power;
	/// FB for halting the axis
	fbHalt: MC_Halt;
	stHaltPrm: ST_AxisHaltParameter;
	/// FB for stopping the axis
	fbStop: MC_Stop;
	stStopPrm: ST_AxisStopParameter;
	/// FB for resetting the axis
	fbReset: MC_Reset;
	/// FB for axis homing
	fbHoming: MC_Home;
	stHomingPrm: ST_AxisHomingParameter;
	/// FB for set axis position
	fbSetPos: MC_SetPosition;
	stSetPosPrm: ST_AxisSetPosParameter;
	/// FB for axis jog
	fbjog: MC_Jog;
	stJogPrm: ST_AxisJogParameter;
	/// FB for axis accelerating jog
	fbJogAcc: MC_MoveVelocity;
	stJogAccPrm: ST_AxisJogAccParameter;
	tonJogAcc: TON;
	/// FB for axis move absolute (this motion command can be overlayed, thus 2 FBs)
	fbMovAbs1: MC_MoveAbsolute;
	fbMovAbs2: MC_MoveAbsolute;
	stMovAbsPrm: ST_AxisMoveAbsParameter;
	/// FB for axis move additive (this motion command can be overlayed, thus 2 FBs)
	fbMovAdd1: MC_MoveAdditive;
	fbMovAdd2: MC_MoveAdditive;
	stMovAddPrm: ST_AxisMoveAddParameter;
	/// FB for axis move relative (this motion command can be overlayed, thus 2 FBs)
	fbMovRel1: MC_MoveRelative;
	fbMovRel2: MC_MoveRelative;
	stMovRelPrm: ST_AxisMoveRelParameter;
	/// FB for axis move modulo (this motion command can be overlayed, thus 2 FBs)
	fbMovMod1: MC_MoveModulo;
	fbMovMod2: MC_MoveModulo;
	stMovModPrm: ST_AxisMoveModParameter;
	/// FB for axis move velocity (this motion command can be overlayed, thus 2 FBs)
	fbMovVel1: MC_MoveVelocity;
	fbMovVel2: MC_MoveVelocity;
	stMovVelPrm: ST_AxisMoveVelParameter;
	/// FB for axis dynamic gear
	fbGearIn: MC_GearInDyn;
	stGearInPrm: ST_AxisGearInParameter;
	fbGearOut: MC_GearOut;
	stGearOutPrm: ST_AxisGearOutParameter;
	
	ii: INT;
	rtrigError: R_TRIG;
	ftrigDiag: F_TRIG;
	///tonTimeOut	: TON;
	tonChkOperation: TON;
	/// ID of the last error in one of the motion FBs
	tonAutoPowerOff: TON;

END_VAR

///
/// Axis driver FB
/// (partly migrated from RMTH FB_MotionCore TwinCAT2)
/// TP/www.rmth.at/10.2014
///

PROPERTY PUBLIC ActModuloPos : LREAL
GET
IF __ISVALIDREF(fbAxisRef) THEN
	ActModuloPos := fbAxisRef.NcToPlc.ModuloActPos;
END_IF
END_GET
END_PROPERTY

PROPERTY PUBLIC ActPos : LREAL
GET
IF __ISVALIDREF(fbAxisRef) THEN
	ActPos := fbAxisRef.NcToPlc.ActPos;
END_IF
END_GET
END_PROPERTY

PROPERTY PUBLIC ActPosEx : LREAL
GET
ActPosEx := stIn.nPositionFeedbackValue*fFeedConstant + fPositionBias;
END_GET
END_PROPERTY

/// Actual amplifier temp. [°C]
PROPERTY AmplifierTemp : LREAL
GET
/// Actual amplifier temp. [°C]
AmplifierTemp := INT_TO_LREAL(stIn.iAmplifierTemperature) / 10;
END_GET
END_PROPERTY

/// Get's the axis reference
PROPERTY Axis : AXIS_REF
GET
Axis := fbAxisRef;
END_GET
END_PROPERTY

PROPERTY AxisId : E_Axis
GET
AxisId := eAxisId;
END_GET
SET
eAxisId := AxisId;
END_SET
END_PROPERTY

/// Get`s the MC axis state.
PROPERTY AxisState : Tc2_MC2.ST_AxisStatus
GET
AxisState := fbAxisRef.Status;
END_GET
END_PROPERTY

PROPERTY AxisType : E_AxisType
GET
AxisType := eAxisType;
END_GET
SET
eAxisType := AxisType;
END_SET
END_PROPERTY

ACTION CheckLatchState:
bLatchedObjPositionOK := ABS(Position - fPosLatched) <= 0.1;
END_ACTION

PROPERTY DefaultParameter : REFERENCE TO ST_AxisDriverParameter
GET
ptDefaultPrm := ADR(stDefaultPrm);
DefaultParameter REF= ptDefaultPrm^;
END_GET
SET
stDefaultPrm := DefaultParameter;
END_SET
END_PROPERTY

PROPERTY Enable : BOOL
GET
Enable := bEnable;
END_GET
SET
bEnable := Enable;
END_SET
END_PROPERTY

PROPERTY EnableLimitSensor : BOOL
GET
EnableLimitSensor := bEnableLimit;
END_GET
SET
bEnableLimit := EnableLimitSensor;
END_SET
END_PROPERTY

PROPERTY EnableNeg : BOOL
GET
EnableNeg:=  bEnableNeg;
END_GET
SET
bEnableNeg:=EnableNeg;
END_SET
END_PROPERTY

PROPERTY EnablePos : BOOL
GET
EnablePos := bEnablePos;
END_GET
SET
bEnablePos := EnablePos;
END_SET
END_PROPERTY

METHOD FB_init : BOOL
VAR_INPUT
	bInitRetains : BOOL; // if TRUE, the retain variables are initialized (warm start / cold start)
	bInCopyCode : BOOL;  // if TRUE, the instance afterwards gets moved into the copy code (online change)
END_VAR
eTyp := E_ComponentType.eComponentType_Axis;
END_METHOD

/// Performs an electronic axis gear-in using default parameter set.
{attribute 'object_name' := 'GearIn'}
METHOD GearIn : E_OperationResult
VAR_INPUT
	/// Gear ratio
	fRatio: LREAL;
	/// Master axis id
	eMasterId: E_Axis;
END_VAR
VAR_IN_OUT
	/// Master axis to gear-in to
	fbMaster: AXIS_REF;
END_VAR
// gear in axis to master

// init result pessimistic
GearIn := E_OperationResult.eOperationResult_NOk;

// if stopping or resetting is active return --> higher prio
IF eCommandExecute = E_MotionCommand.eMotionCommand_reset OR eCommandExecute = E_MotionCommand.eMotionCommand_stop THEN
	RETURN;
END_IF

stGearInPrm := stDefaultPrm.stGearInPrm;
stGearInPrm.fGearRatio := fRatio;
stGearInPrm.eMasterId := eMasterId;
stGearInPrm.fbMaster REF= fbMaster;

eCommandRequest := E_MotionCommand.eMotionCommand_gearIn;
GearIn := E_OperationResult.eOperationResult_Ok;
END_METHOD

/// Performs an electronic axis gear-in using specified parameter
{attribute 'object_name' := 'GearInEx'}
METHOD GearInEx : E_OperationResult
VAR_IN_OUT
	/// Parameter set to use
	stGearInParameter: ST_AxisGearInParameter;
END_VAR
// gear in axis to master

GearInEx := THIS^.GearIn(stGearInParameter.fGearRatio, stGearInParameter.eMasterId, stGearInParameter.fbMaster);

IF GearInEx = E_OperationResult.eOperationResult_Ok THEN
	stGearInPrm := stGearInParameter;
END_IF
END_METHOD

/// Performs an electronic axis gear-out using default parameter set.
{attribute 'object_name' := 'GearOut'}
METHOD GearOut : E_OperationResult
// gear out axis from master

// init result pessimistic
GearOut := E_OperationResult.eOperationResult_NOk;

// if stopping is active return --> higher prio
IF eCommandExecute = E_MotionCommand.eMotionCommand_stop THEN
	RETURN;
END_IF

stGearOutPrm := stDefaultPrm.stGearOutPrm;
eCommandRequest := E_MotionCommand.eMotionCommand_gearOut;
GearOut := E_OperationResult.eOperationResult_Ok;
END_METHOD

/// Performs an electronic axis gear-out using specified parameter
{attribute 'object_name' := 'GearOutEx'}
METHOD GearOutEx : E_OperationResult
VAR_IN_OUT
	/// Parameter set to use
	stGearOutParameter: ST_AxisGearOutParameter;
END_VAR
// gear in axis to master

GearOutEx := THIS^.GearOut();

IF GearOutEx = E_OperationResult.eOperationResult_Ok THEN
	stGearOutPrm := stGearOutParameter;
END_IF
END_METHOD

/// Get's or set's the gear ratio for MC_GearInDyn.
PROPERTY GearRatio : LREAL
GET
// return actual gear ratio
GearRatio := stGearInPrm.fGearRatio;
END_GET
SET
// Updates the gear-ratio (only effective if GearIn was called bevore).
stGearInPrm.fGearRatio := GearRatio;
END_SET
END_PROPERTY

/// Axis halt using default parameter
{attribute 'object_name' := 'Halt'}
METHOD Halt : E_OperationResult
// halt axis

// init result pessimistic
Halt := E_OperationResult.eOperationResult_NOk;

// if stopping is active return --> higher prio: stop
IF eCommandExecute = E_MotionCommand.eMotionCommand_stop THEN
	RETURN;
END_IF

stHaltPrm := stDefaultPrm.stHaltPrm;
//ILog.AddLog('Request received: halt', Concat2('AxisDriver', INT_TO_STRING(THIS^.ID)), E_LogLevel.eLogLevelInformation);
eCommandRequest := E_MotionCommand.eMotionCommand_halt;
Halt := E_OperationResult.eOperationResult_Ok;
END_METHOD

/// Axis halt using specified parameter
{attribute 'object_name' := 'HaltEx'}
METHOD HaltEx : E_OperationResult
VAR_INPUT
	/// Parameter set to use
	stHaltParameter: ST_AxisHaltParameter;
END_VAR
// halt axis

HaltEx := THIS^.Halt();

IF HaltEx = E_OperationResult.eOperationResult_Ok THEN
	stHaltPrm := stHaltParameter;
END_IF
END_METHOD

/// Axis home using default parameter
{attribute 'object_name' := 'Home'}
METHOD Home : E_OperationResult
// home axis

// init result pessimistic
Home := E_OperationResult.eOperationResult_NOk;

// if stopping or resetting is active return --> higher prio
IF eCommandExecute = E_MotionCommand.eMotionCommand_reset OR eCommandExecute = E_MotionCommand.eMotionCommand_stop THEN
	RETURN;
END_IF

stHomingPrm := stDefaultPrm.stHomingPrm;

eCommandRequest := E_MotionCommand.eMotionCommand_home;
Home := E_OperationResult.eOperationResult_Ok;
END_METHOD

PROPERTY Homed : BOOL
GET
Homed:= fbAxisRef.Status.Homed;
END_GET
END_PROPERTY

/// Axis home using specified parameter
{attribute 'object_name' := 'HomeEx'}
METHOD HomeEx : E_OperationResult
VAR_INPUT
	/// Parameter set to use
	stHomingParameter: ST_AxisHomingParameter;
END_VAR
// home axis

HomeEx := THIS^.Home();

IF HomeEx = E_OperationResult.eOperationResult_Ok THEN
	stHomingPrm := stHomingParameter;
END_IF
END_METHOD

PROPERTY Homing : BOOL
GET
Homing:= fbAxisRef.Status.Homing;
END_GET
END_PROPERTY

PROPERTY IsSafetyCardActive : BOOL
GET
VAR
	iTmp: INT;
END_VAR
bSafetyCardAct := FALSE;
FOR iTmp := 0 TO 29 DO
	IF stAX5xxxDiag.stDiagNumberList.arrDiagNumbers[iTmp] = 53506 THEN
		bSafetyCardAct := TRUE;
		EXIT;
	END_IF
END_FOR

IsSafetyCardActive := bSafetyCardAct;
END_GET
END_PROPERTY

/// Axis jog using default parameter
/// This method must be called cyclic (otherwise jog Fwd/Bwd will be reset)
{attribute 'object_name' := 'Jog'}
METHOD Jog : E_OperationResult
VAR_INPUT
	bJogBackwards: BOOL;
	bJogForward: BOOL;
END_VAR
// jog axis

// init result pessimistic
Jog := E_OperationResult.eOperationResult_NOk;

// if stopping or resetting is active return --> higher prio
IF eCommandExecute = E_MotionCommand.eMotionCommand_reset OR eCommandExecute = E_MotionCommand.eMotionCommand_stop THEN
	RETURN;
END_IF

stJogPrm := stDefaultPrm.stJogPrm;
stJogPrm.bJogBackwards := bJogBackwards;
stJogPrm.bJogForward := bJogForward;

IF stJogPrm.bJogBackwards OR stJogPrm.bJogForward THEN
	eCommandRequest := E_MotionCommand.eMotionCommand_jog;
END_IF

Jog := E_OperationResult.eOperationResult_Ok;
END_METHOD

/// Axis jog accelerating using default parameter
/// This method must be called cyclic (otherwise jog Fwd/Bwd will be reset)
{attribute 'object_name' := 'JogAcc'}
METHOD JogAcc : E_OperationResult
VAR_INPUT
	bJogBackwards: BOOL;
	bJogForward: BOOL;
END_VAR
// jog axis acc

// init result pessimistic
JogAcc := E_OperationResult.eOperationResult_NOk;

// if stopping or resetting is active return --> higher prio
IF eCommandExecute = E_MotionCommand.eMotionCommand_reset OR eCommandExecute = E_MotionCommand.eMotionCommand_stop THEN
	RETURN;
END_IF

stJogAccPrm := stDefaultPrm.stJogAccPrm;
stJogAccPrm.bJogBackwards := bJogBackwards;
stJogAccPrm.bJogForward := bJogForward;

IF stJogAccPrm.bJogBackwards OR stJogAccPrm.bJogForward THEN
	eCommandRequest := E_MotionCommand.eMotionCommand_jogAcc;
END_IF

JogAcc := E_OperationResult.eOperationResult_Ok;
END_METHOD

/// Axis jog accelerating using specified parameter
{attribute 'object_name' := 'JogAccEx'}
METHOD JogAccEx : E_OperationResult
VAR_INPUT
	/// Parameter set to use
	stJogAccParameter: ST_AxisJogAccParameter;
END_VAR
// jog acc axis

JogAccEx := THIS^.JogAcc(stJogAccParameter.bJogBackwards, stJogAccParameter.bJogForward);

IF JogAccEx = E_OperationResult.eOperationResult_Ok THEN
	stJogAccPrm := stJogAccParameter;
END_IF
END_METHOD

/// Axis jog accelerating using default parameter
/// This method must be called cyclic (otherwise jog Fwd/Bwd will be reset)
{attribute 'object_name' := 'JogAccExVel'}
METHOD JogAccExVel : E_OperationResult
VAR_INPUT
	bJogBackwards: BOOL;
	bJogForward: BOOL;
	/// Slow (starting) speed
	fSlowSpeed: LREAL;
	/// Fast end-speed
	fFastSpeed: LREAL;
	/// Time for ramp from slow to fast speed [ms]
	fAccTime: LREAL;
END_VAR
// jog axis acc

// init result pessimistic
JogAccExVel := E_OperationResult.eOperationResult_NOk;

// if stopping or resetting is active return --> higher prio
IF eCommandExecute = E_MotionCommand.eMotionCommand_reset OR eCommandExecute = E_MotionCommand.eMotionCommand_stop THEN
	RETURN;
END_IF

stJogAccPrm := stDefaultPrm.stJogAccPrm;
stJogAccPrm.fSlowSpeed := fSlowSpeed;
stJogAccPrm.fFastSpeed := fFastSpeed;
stJogAccPrm.tAccTime := LREAL_TO_TIME(fAccTime);
stJogAccPrm.bJogBackwards := bJogBackwards;
stJogAccPrm.bJogForward := bJogForward;

IF stJogAccPrm.bJogBackwards OR stJogAccPrm.bJogForward THEN
	eCommandRequest := E_MotionCommand.eMotionCommand_jogAcc;
END_IF

JogAccExVel := E_OperationResult.eOperationResult_Ok;
END_METHOD

/// Axis jog using specified parameter
{attribute 'object_name' := 'JogEx'}
METHOD JogEx : E_OperationResult
VAR_INPUT
	/// Parameter set to use
	stJogParameter: ST_AxisJogParameter;
END_VAR
// jog axis

JogEx := THIS^.Jog(stJogParameter.bJogBackwards, stJogParameter.bJogForward);

IF JogEx = E_OperationResult.eOperationResult_Ok THEN
	stJogPrm := stJogParameter;
END_IF
END_METHOD

/// Axis jog using specified parameter
{attribute 'object_name' := 'JogExVel'}
METHOD JogExVel : E_OperationResult
VAR_INPUT
	bJogBackwards: BOOL;
	bJogForward: BOOL;
	/// Velocity
	fVelocity: LREAL;
	/// Modus
	eMode: E_JogMode := E_JogMode.MC_JOGMODE_INCHING;
END_VAR
// jog axis

JogExVel := THIS^.Jog(bJogBackwards, bJogForward);

IF JogExVel = E_OperationResult.eOperationResult_Ok THEN
	stJogPrm := stDefaultPrm.stJogPrm;
	stJogPrm.eMode := eMode;
	stJogPrm.fVelocity := fVelocity;
	stJogPrm.bJogBackwards := bJogBackwards;
	stJogPrm.bJogForward := bJogForward;
END_IF
END_METHOD

PROPERTY LastMcErrorId : UDINT
GET
LastMcErrorId := nErrorID;
END_GET
END_PROPERTY

METHOD LatchObjState : BOOL
VAR_INPUT
END_VAR
fPosLatched := Position;
END_METHOD

PROPERTY LimitNeg : LREAL
GET
LimitNeg := nLimitNeg;
END_GET
SET
nLimitNeg := LimitNeg;
END_SET
END_PROPERTY

PROPERTY LimitPos : LREAL
GET
LimitPos := nLimitPos;
END_GET
SET
nLimitPos := LimitPos;
END_SET
END_PROPERTY

PROPERTY MasterAxisId : E_Axis
GET
MasterAxisId := eMasterAxisId;
END_GET
END_PROPERTY

PROPERTY MotionState : MC_AxisStates
GET
MotionState := fbAxisRef.Status.MotionState;
END_GET
END_PROPERTY

/// Actual motor temp. [°C]
PROPERTY MotorTemp : LREAL
GET
/// Actual motor temp. [°C]
MotorTemp := INT_TO_LREAL(stIn.iMotorTemperature) / 10;
END_GET
END_PROPERTY

/// Performs an absolute axis positioning using default parameter set.
/// This motion is capable to overlay (max. 2 parallel at one time)
{attribute 'object_name' := 'MoveAbs'}
METHOD MoveAbs : E_OperationResult
VAR_INPUT
	/// Position to move to
	fPosition: LREAL;
END_VAR
// move axis abs

// init result pessimistic
MoveAbs := E_OperationResult.eOperationResult_NOk;

// if stopping or resetting is active return --> higher prio
IF eCommandExecute = E_MotionCommand.eMotionCommand_reset OR eCommandExecute = E_MotionCommand.eMotionCommand_stop THEN
	RETURN;
END_IF

stMovAbsPrm := stDefaultPrm.stMovAbsPrm;
stMovAbsPrm.fPosition := fPosition;

fPosRequest:=  fPosition;
eCommandRequest := E_MotionCommand.eMotionCommand_moveAbs;
MoveAbs := E_OperationResult.eOperationResult_Ok;
END_METHOD

/// Performs an absolute axis positioning using specified parameter
/// This motion is capable to overlay (max. 2 parallel at one time)
{attribute 'object_name' := 'MoveAbsEx'}
METHOD MoveAbsEx : E_OperationResult
VAR_INPUT
	/// Parameter set to use
	stMovAbsParameter: ST_AxisMoveAbsParameter;
END_VAR
// move axis abs

MoveAbsEx := THIS^.MoveAbs(stMovAbsParameter.fPosition);

IF MoveAbsEx = E_OperationResult.eOperationResult_Ok THEN
	stMovAbsPrm := stMovAbsParameter;
END_IF
END_METHOD

/// Performs an absolute axis positioning using input parameter set.
/// This motion is capable to overlay (max. 2 parallel at one time)
{attribute 'object_name' := 'MoveAbsExVel'}
METHOD MoveAbsExVel : E_OperationResult
VAR_INPUT
	/// Position to move to
	fPosition: LREAL;
	/// Speed
	fVelocity: LREAL;
END_VAR
// move axis abs

// init result pessimistic
MoveAbsExVel := E_OperationResult.eOperationResult_NOk;

// if stopping or resetting is active return --> higher prio
IF eCommandExecute = E_MotionCommand.eMotionCommand_reset OR eCommandExecute = E_MotionCommand.eMotionCommand_stop THEN
	RETURN;
END_IF

stMovAbsPrm := stDefaultPrm.stMovAbsPrm;
stMovAbsPrm.fPosition := fPosition;
stMovAbsPrm.fVelocity := fVelocity;

fPosRequest:=  fPosition;

eCommandRequest := E_MotionCommand.eMotionCommand_moveAbs;
MoveAbsExVel := E_OperationResult.eOperationResult_Ok;
END_METHOD

/// Performs an additive axis positioning using default parameter set.
/// This motion is capable to overlay (max. 2 parallel at one time)
{attribute 'object_name' := 'MoveAdd'}
METHOD MoveAdd : E_OperationResult
VAR_INPUT
	/// Distance
	fDistance: LREAL;
END_VAR
// move axis add

// init result pessimistic
MoveAdd := E_OperationResult.eOperationResult_NOk;

// if stopping or resetting is active return --> higher prio
IF eCommandExecute = E_MotionCommand.eMotionCommand_reset OR eCommandExecute = E_MotionCommand.eMotionCommand_stop THEN
	RETURN;
END_IF

stMovAddPrm := stDefaultPrm.stMovAddPrm;
stMovAddPrm.fDistance := fDistance;

fPosRequest:=  fbAxisRef.NcToPlc.ActPos+fDistance;

eCommandRequest := E_MotionCommand.eMotionCommand_moveAdd;
MoveAdd := E_OperationResult.eOperationResult_Ok;
END_METHOD

/// Performs an additive axis positioning using specified parameter set.
/// This motion is capable to overlay (max. 2 parallel at one time)
{attribute 'object_name' := 'MoveAddEx'}
METHOD MoveAddEx : E_OperationResult
VAR_INPUT
	/// Parameter set to use
	stMovAddParameter: ST_AxisMoveAddParameter;
END_VAR
// move axis add

MoveAddEx := THIS^.MoveAdd(stMovAddParameter.fDistance);

IF MoveAddEx = E_OperationResult.eOperationResult_Ok THEN
	stMovAddPrm := stMovAddParameter;
END_IF
END_METHOD

/// Performs an modulo axis positioning using default parameter set.
/// This motion is capable to overlay (max. 2 parallel at one time)
{attribute 'object_name' := 'MoveMod'}
METHOD MoveMod : E_OperationResult
VAR_INPUT
	/// Position to move to
	fPosition: LREAL;
END_VAR
// move axis mod

// init result pessimistic
MoveMod := E_OperationResult.eOperationResult_NOk;

// if stopping or resetting is active return --> higher prio
IF eCommandExecute = E_MotionCommand.eMotionCommand_reset OR eCommandExecute = E_MotionCommand.eMotionCommand_stop THEN
	RETURN;
END_IF

stMovModPrm := stDefaultPrm.stMovModPrm;
stMovModPrm.fPosition := fPosition;

fPosRequest:=  fPosition;
eCommandRequest := E_MotionCommand.eMotionCommand_moveMod;
MoveMod := E_OperationResult.eOperationResult_Ok;
END_METHOD

/// Performs an modulo axis positioning using specified parameter
/// This motion is capable to overlay (max. 2 parallel at one time)
{attribute 'object_name' := 'MoveModEx'}
METHOD MoveModEx : E_OperationResult
VAR_INPUT
	/// Parameter set to use
	stMovModParameter: ST_AxisMoveModParameter;
END_VAR
// move axis mod

MoveModEx := THIS^.MoveMod(stMovModParameter.fPosition);

IF MoveModEx = E_OperationResult.eOperationResult_Ok THEN
	stMovModPrm := stMovModParameter;
END_IF
END_METHOD

/// Performs an relative axis positioning using default parameter set.
/// This motion is capable to overlay (max. 2 parallel at one time)
{attribute 'object_name' := 'MoveRel'}
METHOD MoveRel : E_OperationResult
VAR_INPUT
	/// Distance
	fDistance: LREAL;
END_VAR
// move axis rel

// init result pessimistic
MoveRel := E_OperationResult.eOperationResult_NOk;

// if stopping or resetting is active return --> higher prio
IF eCommandExecute = E_MotionCommand.eMotionCommand_reset OR eCommandExecute = E_MotionCommand.eMotionCommand_stop THEN
	RETURN;
END_IF

stMovRelPrm := stDefaultPrm.stMovRelPrm;
stMovRelPrm.fDistance := fDistance;

fPosRequest:=  fbAxisRef.NcToPlc.ActPos+fDistance;

eCommandRequest := E_MotionCommand.eMotionCommand_moveRel;
MoveRel := E_OperationResult.eOperationResult_Ok;
END_METHOD

/// Performs an relative axis positioning using specified parameter set.
/// This motion is capable to overlay (max. 2 parallel at one time)
{attribute 'object_name' := 'MoveRelEx'}
METHOD MoveRelEx : E_OperationResult
VAR_INPUT
	/// Parameter set to use
	stMovRelParameter: ST_AxisMoveRelParameter;
END_VAR
// move axis rel

MoveRelEx := THIS^.MoveRel(stMovRelParameter.fDistance);

IF MoveRelEx = E_OperationResult.eOperationResult_Ok THEN
	stMovRelPrm := stMovRelParameter;
END_IF
END_METHOD

/// Performs an relative axis positioning using specified parameter set.
/// This motion is capable to overlay (max. 2 parallel at one time)
{attribute 'object_name' := 'MoveRelExVel'}
METHOD MoveRelExVel : E_OperationResult
VAR_INPUT
	/// Distance to move to
	fDistance: LREAL;
	/// Speed
	fVelocity: LREAL;
END_VAR
// move axis rel

// init result pessimistic
MoveRelExVel := E_OperationResult.eOperationResult_NOk;

// if stopping or resetting is active return --> higher prio
IF eCommandExecute = E_MotionCommand.eMotionCommand_reset OR eCommandExecute = E_MotionCommand.eMotionCommand_stop THEN
	RETURN;
END_IF

stMovRelPrm := stDefaultPrm.stMovRelPrm;
stMovRelPrm.fDistance := fDistance;
stMovRelPrm.fVelocity := fVelocity;

fPosRequest:=  fbAxisRef.NcToPlc.ActPos+fDistance;

eCommandRequest := E_MotionCommand.eMotionCommand_moveRel;
MoveRelExVel := E_OperationResult.eOperationResult_Ok;
END_METHOD

/// Performs an velocity axis movement using default parameter set.
/// This motion is capable to overlay (max. 2 parallel at one time)
{attribute 'object_name' := 'MoveVel'}
METHOD MoveVel : E_OperationResult
VAR_INPUT
	/// Velocity
	fVelocity: LREAL;
	/// Direction
	eDirection: MC_Direction;
END_VAR
// move axis vel

// init result pessimistic
MoveVel := E_OperationResult.eOperationResult_NOk;

// if stopping or resetting is active return --> higher prio
IF eCommandExecute = E_MotionCommand.eMotionCommand_reset OR eCommandExecute = E_MotionCommand.eMotionCommand_stop THEN
	RETURN;
END_IF

stMovVelPrm := stDefaultPrm.stMovVelPrm;
stMovVelPrm.fVelocity := fVelocity;
stMovVelPrm.eDirection := eDirection;

eCommandRequest := E_MotionCommand.eMotionCommand_moveVel;
MoveVel := E_OperationResult.eOperationResult_Ok;
END_METHOD

/// Performs an velocity axis movement using specified parameter
/// This motion is capable to overlay (max. 2 parallel at one time)
{attribute 'object_name' := 'MoveVelEx'}
METHOD MoveVelEx : E_OperationResult
VAR_INPUT
	/// Parameter set to use
	stMovVelParameter: ST_AxisMoveVelParameter;
END_VAR
// move axis abs

MoveVelEx := THIS^.MoveVel(stMovVelParameter.fVelocity, stMovVelParameter.eDirection);

IF MoveVelEx = E_OperationResult.eOperationResult_Ok THEN
	stMovVelPrm := stMovVelParameter;
END_IF
END_METHOD

PROPERTY Moving : BOOL
GET
Moving := fbAxisRef.Status.Moving;
END_GET
END_PROPERTY

/// The torque limit for both directions. [Nm]
PROPERTY negTorqueLimit : LREAL
GET
/// The torque limit for both directions. [1/10%]
negTorqueLimit := INT_TO_LREAL(stOut.iNegativeTorqueLimitValue) * stDefaultPrm.stGeneralPrm.fTorqueFactor;
END_GET
SET
stOut.iNegativeTorqueLimitValue := ABS(LREAL_TO_INT(negTorqueLimit/stDefaultPrm.stGeneralPrm.fTorqueFactor));
END_SET
END_PROPERTY

PROPERTY NotMoving : BOOL
GET
NotMoving := fbAxisRef.Status.NotMoving;
END_GET
END_PROPERTY

PROPERTY Override : LREAL
GET
Override := fbPower.Override;
END_GET
SET
fbPower.Override := Override;
END_SET
END_PROPERTY

/// The torque limit for both directions. [Nm]
PROPERTY posTorqueLimit : LREAL
GET
/// The torque limit for both directions. [1/10%]
posTorqueLimit := INT_TO_LREAL(stOut.iPositiveTorqueLimitValue) * stDefaultPrm.stGeneralPrm.fTorqueFactor;
END_GET
SET
stOut.iPositiveTorqueLimitValue := ABS(LREAL_TO_INT(posTorqueLimit/stDefaultPrm.stGeneralPrm.fTorqueFactor));
END_SET
END_PROPERTY

/// Reset component logic
{attribute '' := ''}
{attribute 'object_name' := 'Reset'}
METHOD Reset
// base logic run
SUPER^.Reset();

// reset axis
eCommandRequest := E_MotionCommand.eMotionCommand_reset;
eState := E_ComponentState.eComponentState_resetting;
END_METHOD

/// Run component logic
{attribute 'object_name' := 'Run'}
METHOD Run : E_ComponentState
// base logic run
Run := SUPER^.Run();

// return here as long axis ref not set
IF NOT __ISVALIDREF(fbAxisRef) THEN
	sClearText := 'Axis ref not set!';
	RETURN;
END_IF

// switch case request
CASE eCommandRequest OF	
	/// No command
	E_MotionCommand.eMotionCommand_none:
	
	/// Reset axis
	E_MotionCommand.eMotionCommand_reset:
		IF (eCommandExecute <> E_MotionCommand.eMotionCommand_stop AND eCommandExecute <> E_MotionCommand.eMotionCommand_halt) OR fbAxisRef.Status.StandStill THEN
			eCommandExecute := eCommandRequest;
			eCommandRequest := E_MotionCommand.eMotionCommand_none;
		END_IF
	
	/// Axis halt (default stopping method)
	E_MotionCommand.eMotionCommand_halt:
		IF eCommandExecute <> E_MotionCommand.eMotionCommand_stop THEN
			eCommandExecute := eCommandRequest;
			eCommandRequest := E_MotionCommand.eMotionCommand_none;
		END_IF;
	
	/// Axis stop (needs reset before next motion command)
	E_MotionCommand.eMotionCommand_stop:
		eCommandExecute := eCommandRequest;
		eCommandRequest := E_MotionCommand.eMotionCommand_none;
	
	/// other commands
	E_MotionCommand.eMotionCommand_home,
	E_MotionCommand.eMotionCommand_setPos,
	E_MotionCommand.eMotionCommand_jog,
	E_MotionCommand.eMotionCommand_jogAcc,
	E_MotionCommand.eMotionCommand_moveAbs,
	E_MotionCommand.eMotionCommand_moveAdd,
	E_MotionCommand.eMotionCommand_moveRel,
	E_MotionCommand.eMotionCommand_moveMod,
	E_MotionCommand.eMotionCommand_moveVel,
	E_MotionCommand.eMotionCommand_torque,
	E_MotionCommand.eMotionCommand_gearIn,
	E_MotionCommand.eMotionCommand_gearOut,
	E_MotionCommand.eMotionCommand_touchProbe:
		// wait for active command none and axis ready
		IF eCommandExecute = eMotionCommand_none THEN
			eCommandExecute := eCommandRequest;
			eCommandRequest := E_MotionCommand.eMotionCommand_none;
		ELSE
			eCommandRequest := E_MotionCommand.eMotionCommand_none;
		END_IF
END_CASE

// call workflows 
WfDiagnostic();
WfPower();
WfReset();
WfHome();
WfSetPos();
WfJog();
WfJogAcc();
WfMovAbs();
WfMovAdd();
WfMovRel();
WfMovMod();
WfMovVel();
WfGearIn();
WfGearOut();
WfHalt();
WfStop();
WfErrorHandling();

// set clear text
IF eState <> E_ComponentState.eComponentState_error THEN
	sClearText := SEL(fbAxisRef.Status.Operational, 'Antrieb nicht aktiviert!', Concat('Antrieb Status: ', StateAsString));
ELSE
	sClearText := Concat('Fehler Antrieb, FehlerNr: ', UDINT_TO_STRING(nErrorID));
	// try get details
	IF eAxisType = E_AxisType.AX5xxx THEN
		sMsg := stAX5xxxDiag.strDiagMessage; // display diag msg
		FOR ii := 0 TO 2 DO	// add first 3 error codes 
			sMsg := Concat3(sMsg, ', ', UDINT_TO_STRING(stAX5xxxDiag.stDiagNumberList.arrDiagNumbers[ii]));
		END_FOR
		sClearText := sMsg;
	END_IF
END_IF

// Ausgabedaten
Error := (eState = E_ComponentState.eComponentState_error);
Position := fbAxisRef.NcToPlc.ActPos;

CheckLatchState();
END_METHOD

/// Set axis reference
{attribute 'object_name' := 'SetAxisReference'}
METHOD SetAxisReference
VAR_IN_OUT
	/// NC Axis reference
	fbRefAxis: AXIS_REF;
	/// Additional inputs from axis
	stRefIn: ST_AxisIn;
	/// Additional outputs to axis
	stRefOut: ST_AxisOut;
END_VAR
fbAxisRef REF= fbRefAxis;
stIn REF= stRefIn;
stOut REF= stRefOut;

DefaultParameter.stHomingPrm.bCalibrationCam REF= stIn.bCalibrationCam;
END_METHOD

/// Set axis position
{attribute 'object_name' := 'SetPos'}
METHOD SetPos : E_OperationResult
VAR_INPUT
	fPosition: LREAL;
END_VAR
// set axis pos

// init result pessimistic
SetPos := E_OperationResult.eOperationResult_NOk;

// if stopping or resetting is active return --> higher prio
IF eCommandExecute = E_MotionCommand.eMotionCommand_reset OR eCommandExecute = E_MotionCommand.eMotionCommand_stop THEN
	RETURN;
END_IF

stSetPosPrm := stDefaultPrm.stSetPosPrm;
stSetPosPrm.fPosition := fPosition;

eCommandRequest := E_MotionCommand.eMotionCommand_setPos;
SetPos := E_OperationResult.eOperationResult_Ok;
END_METHOD

/// Set axis position, extended method with all options
{attribute 'object_name' := 'SetPosEx'}
METHOD SetPosEx : E_OperationResult
VAR_INPUT
	/// Parameter set to use
	stSetPosParameter: ST_AxisSetPosParameter;
END_VAR
// set axis pos

SetPosEx := THIS^.SetPos(stSetPosParameter.fPosition);

IF SetPosEx = E_OperationResult.eOperationResult_Ok THEN
	stSetPosPrm := stSetPosParameter;
END_IF
END_METHOD

METHOD SetSecondPosFeedback
VAR_INPUT	
	PositionBias	: LREAL;
	FeedConstant	: LREAL;
END_VAR
fPositionBias := PositionBias;
fFeedConstant := FeedConstant;
END_METHOD

/// Axis stop using default parameter
{attribute 'object_name' := 'Stop'}
METHOD Stop : E_OperationResult
// stop axis

stStopPrm := stDefaultPrm.stStopPrm;

eCommandRequest := E_MotionCommand.eMotionCommand_stop;
Stop := E_OperationResult.eOperationResult_Ok;
END_METHOD

/// Axis stop using specified parameter
{attribute 'object_name' := 'StopEx'}
METHOD StopEx : E_OperationResult
VAR_INPUT
	/// Parameter set to use
	stStopParameter: ST_AxisStopParameter;
END_VAR
// stop axis

StopEx := THIS^.Stop();
stStopPrm := stStopParameter;
END_METHOD

METHOD TargetReached : BOOL
VAR_INPUT
	fWindow: LREAL;
END_VAR
TargetReached := ABS(fbAxisRef.NcToPlc.Actpos - fPosRequest) < fWindow;
END_METHOD

METHOD TargetReachedMod : BOOL
VAR_INPUT
	fWindow: LREAL;
END_VAR
TargetReachedMod := ABS(fbAxisRef.NcToPlc.ModuloActPos - fPosRequest) < fWindow;
END_METHOD

/// Actual torque [Nm]
PROPERTY Torque : LREAL
GET
/// Actual torque [Nm]
Torque := INT_TO_LREAL(stIn.iTorqueFeedbackValue) * stDefaultPrm.stGeneralPrm.fTorqueFactor;
END_GET
END_PROPERTY

/// The torque limit for both directions. [Nm]
PROPERTY TorqueLimit : LREAL
GET
/// The torque limit for both directions. [1/10%]
TorqueLimit := INT_TO_LREAL(stOut.iBipolarTorqueLimitValue) * stDefaultPrm.stGeneralPrm.fTorqueFactor;
END_GET
SET
stOut.iBipolarTorqueLimitValue := ABS(LREAL_TO_INT(TorqueLimit/stDefaultPrm.stGeneralPrm.fTorqueFactor));
END_SET
END_PROPERTY

PROPERTY Velocity : LREAL
GET
IF __ISVALIDREF(fbAxisRef) THEN
	Velocity  := fbAxisRef.NcToPlc.ActVelo;	
END_IF
END_GET
END_PROPERTY

ACTION WfDiagnostic:

/// Workflow axis diagnostic

// run axis FBs
fbAxisRef.ReadStatus();

// return in case of reset
(*IF eCommandExecute = E_MotionCommand.eMotionCommand_reset THEN
	RETURN;
END_IF*)

// diagnostics AX5xxx
IF eAxisType = E_AxisType.AX5xxx THEN
	// Diag + Reset of AX5000
	// call drive diag FBs
	fbAX5xxxDiag(
		IPCNetID	:= IPCNetID,
		Axis		:= fbAxisRef,
		stAX5000Diag:= stAX5xxxDiag);

	// clear reset/diag request if not active
	fbAX5xxxDiag.Reset := fbAX5xxxDiag.Reset AND fbAX5xxxDiag.ResetAct;
	fbAX5xxxDiag.GetDiag := fbAX5xxxDiag.GetDiag AND fbAX5xxxDiag.DiagAct;

	//IF fbAX5xxxDiag.Error THEN... / nErrorId := fbAX5xxxDiag.AdsErrId; -> WfErrorHandling
	stDriveRef := fbAX5xxxDiag.DriveRef;
END_IF
END_ACTION

ACTION WfErrorHandling:
// chk axis operational
tonChkOperation(IN := (eState = E_ComponentState.eComponentState_running AND fbPower.Enable AND NOT fbAxisRef.Status.Operational), PT := T#5S);
IF tonChkOperation.Q THEN
	eState := E_ComponentState.eComponentState_error;
END_IF

// run error trigger
rtrigError(CLK := fbAxisRef.Status.Error OR stAX5xxxDiag.bAxisError OR eState = E_ComponentState.eComponentState_error);
IF rtrigError.Q THEN
	eState := E_ComponentState.eComponentState_error;
	IF eAxisType = E_AxisType.AX5xxx THEN
		bErrDiagActive := TRUE;	
		fbAX5xxxDiag.GetDiag := TRUE; // get diag for AX5xxx
	ELSE
		WriteError(E_Event.eEvent_none ,Concat4('Fehler Antrieb ', Name, ', FehlerNr: ', UDINT_TO_STRING(nErrorId)));
	END_IF
END_IF

// run AX5000 diag 
ftrigDiag(CLK := fbAX5xxxDiag.DiagAct);
IF ftrigDiag.Q AND bErrDiagActive THEN
	bErrDiagActive := FALSE;
	IF fbAxisRef.Status.Error OR IsSafetyCardActive THEN // HW error
		IF bSafetyCardAct THEN
			sMsg := Concat(Name, ': Safety Card aktiv'); // display diag msg
		ELSE
			sMsg := Concat3(Name, ': ', stAX5xxxDiag.strDiagMessage); // display diag msg
			FOR ii := 0 TO 2 DO	// add first 3 error codes 
				sMsg := Concat3(sMsg, ', ', UDINT_TO_STRING(stAX5xxxDiag.stDiagNumberList.arrDiagNumbers[ii]));
			END_FOR
		END_IF		
		WriteError(E_Event.eEvent_none , sMsg);		

	ELSE
		sMsg := Concat4('Achse ', INT_TO_STRING(eAxisId), ': ', sLastError);
		sMsg := Concat3(sMsg, ' / FehlerNr: ', UDINT_TO_STRING(nErrorId));
		WriteError(E_Event.eEvent_none , sMsg);			
	END_IF
END_IF;
END_ACTION

ACTION WfGearIn:

/// Workflow gear in

// call fb cyclic
fbGearIn.GearRatio := stGearInPrm.fGearRatio;
fbGearIn.Acceleration := stGearInPrm.fAcceleration;
fbGearIn.Deceleration := stGearInPrm.fDeceleration;
fbGearIn.Jerk := stGearInPrm.fJerk;
fbGearIn.BufferMode := stGearInPrm.eBufferMode;
fbGearIn.Options := stGearInPrm.stOptions;
IF __ISVALIDREF(stGearInPrm.fbMaster) THEN
	fbGearIn(Master := stGearInPrm.fbMaster, Slave := fbAxisRef);	
END_IF

// FB diagnostic and reset 
IF fbGearIn.Enable AND NOT fbGearIn.Busy THEN
	IF fbGearIn.Error THEN			
		nErrorId := fbGearIn.ErrorID;
		sLastError := 'Fehler Antrieb Koppeln.';
		eState := E_ComponentState.eComponentState_error;			
	END_IF
	fbGearIn.Enable := FALSE;
END_IF

// set master axis ID
eMasterAxisId := SEL(fbAxisRef.Status.Coupled, eAxisId, stGearInPrm.eMasterId);

// return if other command active	
IF eCommandExecute <> E_MotionCommand.eMotionCommand_gearIn THEN
	RETURN;
END_IF

sClearText := 'Antrieb Koppeln';		
IF NOT fbGearIn.InGear THEN
	fbGearIn.Enable := TRUE;
END_IF
eCommandExecute := E_MotionCommand.eMotionCommand_none;
END_ACTION

ACTION WfGearOut:

/// Workflow gear out

// call fb cyclic
fbGearOut.Options := stGearOutPrm.stOptions;
fbGearOut(Slave := fbAxisRef);

// FB diagnostic and reset 
IF fbGearOut.Execute AND NOT fbGearOut.Busy THEN
	IF fbGearOut.Error THEN
		nErrorId := fbGearOut.ErrorID;
		sLastError := 'Fehler Antrieb Entkoppeln.';
		eState := E_ComponentState.eComponentState_error;			
	END_IF
	fbGearOut.Execute := FALSE;
END_IF
		
// return if not in gear out
IF eCommandExecute <> E_MotionCommand.eMotionCommand_gearOut THEN
	RETURN;
END_IF

sClearText := 'Antrieb Entoppeln';
IF stGearOutPrm.bHaltAxis THEN
	stHaltPrm.eBufferMode := MC_Aborting;
	stHaltPrm.fDeceleration := stGearInPrm.fDeceleration;
	stHaltPrm.fJerk := stGearInPrm.fJerk;
	//stHaltPrm.stOptions := stGearInPrm.stOptions;
	THIS^.HaltEx(stHaltPrm);
ELSE
	fbGearOut(Slave := fbAxisRef, Execute := TRUE);	
END_IF
eCommandExecute := E_MotionCommand.eMotionCommand_none;
END_ACTION

ACTION WfHalt:

/// Workflow halting

// call fb cyclic
fbHalt.BufferMode := stHaltPrm.eBufferMode;
fbHalt.Deceleration := stHaltPrm.fDeceleration;
fbHalt.Jerk := stHaltPrm.fJerk;
fbHalt.Options := stHaltPrm.stOptions;
fbHalt(Axis := fbAxisRef);

// FB diagnostic and reset 
IF fbHalt.Execute AND NOT fbHalt.Busy THEN
	IF fbHalt.Error THEN
		nErrorId := fbHalt.ErrorID;
		sLastError := 'Fehler bei Antrieb Halt.';
		eState := E_ComponentState.eComponentState_error;			
	END_IF
	fbHalt.Execute := FALSE;
END_IF
		
// return if not in halting
IF eCommandExecute <> E_MotionCommand.eMotionCommand_halt THEN
	RETURN;
END_IF

sClearText := 'Antrieb Halt';
fbHalt(Axis := fbAxisRef, Execute := TRUE);
eCommandExecute := E_MotionCommand.eMotionCommand_none;
IF fbAxisRef.Status.StandStill THEN
	eCommandExecute := E_MotionCommand.eMotionCommand_none;
END_IF
END_ACTION

ACTION WfHome:

/// Workflow homing

// call fb cyclic
fbHoming.bCalibrationCam := SEL(__ISVALIDREF(stHomingPrm.bCalibrationCam), FALSE, stHomingPrm.bCalibrationCam);
fbHoming.BufferMode := stHomingPrm.eBufferMode;
fbHoming.HomingMode := stHomingPrm.eHomingMode;
fbHoming.Options := stHomingPrm.stOptions;
fbHoming.Position := stHomingPrm.fPosition;
fbHoming(Axis := fbAxisRef);

// FB diagnostic and reset 
IF fbHoming.Execute AND NOT fbHoming.Busy THEN
	IF fbHoming.Error THEN
		nErrorId := fbHoming.ErrorID;
		sLastError := 'Fehler Antrieb GRST';
		eState := E_ComponentState.eComponentState_error;			
	END_IF
	fbHoming.Execute := FALSE;
END_IF
		
// return if not in homing
IF eCommandExecute <> E_MotionCommand.eMotionCommand_home THEN
	RETURN;
END_IF

sClearText := 'Antrieb GRST';		
IF NOT fbHoming.Busy THEN
	fbHoming(Axis := fbAxisRef, Execute := TRUE);
	eCommandExecute := E_MotionCommand.eMotionCommand_none;
END_IF
END_ACTION

ACTION WfJog:

/// Workflow jog axis

// call fb cyclic
fbjog.JogBackwards := stJogPrm.bJogBackwards;
fbjog.JogForward := stJogPrm.bJogForward;
fbjog.Acceleration := stJogPrm.fAcceleration;
fbjog.Deceleration := stJogPrm.fDeceleration;
fbjog.Jerk := stJogPrm.fJerk;
fbjog.Mode := stJogPrm.eMode;
fbjog.Position := stJogPrm.fPosition;
fbjog.Velocity := stJogPrm.fVelocity;
fbjog(Axis := fbAxisRef);

// reset jog F/B each cycle (stop's axis if Jog/JogEx method isn't called anymore)
stJogPrm.bJogBackwards := FALSE;
stJogPrm.bJogForward := FALSE;

// return if not in jog
IF eCommandExecute <> E_MotionCommand.eMotionCommand_jog THEN
	RETURN;
END_IF

// case of jog error
IF fbjog.Error  THEN
	nErrorId := fbjog.ErrorID;
	sLastError := 'Fehler Antrieb Tippen.';
	eState := E_ComponentState.eComponentState_error;			
END_IF		

eCommandExecute := E_MotionCommand.eMotionCommand_none;
END_ACTION

ACTION WfJogAcc:

/// Workflow jog axis acc

// call fb's cyclic
fbJogAcc.Direction := MC_Current_Direction;
fbJogAcc.Direction := SEL(stJogAccPrm.bJogForward, MC_Negative_Direction, MC_Positive_Direction);
fbJogAcc.Acceleration := stJogAccPrm.fAcceleration;
fbJogAcc.Deceleration := stJogAccPrm.fDeceleration;
fbJogAcc.Jerk := stJogAccPrm.fJerk;
fbJogAcc.BufferMode := stJogAccPrm.eBufferMode;
fbJogAcc.Options := stJogAccPrm.stOptions;
fbJogAcc(Axis := fbAxisRef);

